  PROC DrawPart72()
    MoveL Offs(pOrigin,295.05,63.65,0.00),v40,z0,tPen\WObj:=wPaper;
    MoveL Offs(pOrigin,298.24,62.80,0.00),v40,z0,tPen\WObj:=wPaper;
    MoveL Offs(pOrigin,301.21,64.85,0.00),v40,z0,tPen\WObj:=wPaper;
    MoveL Offs(pOrigin,304.83,66.20,0.00),v40,z0,tPen\WObj:=wPaper;
    MoveL Offs(pOrigin,310.14,67.40,0.00),v40,z0,tPen\WObj:=wPaper;
    MoveL Offs(pOrigin,314.17,69.95,0.00),v40,z0,tPen\WObj:=wPaper;
    MoveL Offs(pOrigin,316.73,70.95,0.00),v40,z0,tPen\WObj:=wPaper;
    MoveL Offs(pOrigin,322.46,72.57,0.00),v40,z0,tPen\WObj:=wPaper;
    MoveL Offs(pOrigin,333.30,74.49,0.00),v40,z0,tPen\WObj:=wPaper;
    MoveL Offs(pOrigin,334.15,74.91,0.00),v40,z0,tPen\WObj:=wPaper;
    MoveL Offs(pOrigin,334.15,74.91,0.00),v40,z0,tPen\WObj:=wPaper;
    MoveL Offs(pOrigin,340.17,88.09,0.00),v40,z0,tPen\WObj:=wPaper;
    MoveL Offs(pOrigin,342.01,92.97,0.00),v40,z0,tPen\WObj:=wPaper;
    MoveL Offs(pOrigin,341.09,93.74,0.00),v40,z0,tPen\WObj:=wPaper;
    MoveL Offs(pOrigin,345.30,89.53,0.00),v40,z0,tPen\WObj:=wPaper;
    MoveL Offs(pOrigin,344.92,89.84,0.00),v40,z0,tPen\WObj:=wPaper;
    MoveL Offs(pOrigin,341.77,86.69,0.00),v40,fine,tPen\WObj:=wPaper;
    MoveL Offs(pOrigin,341.77,86.69,6.00),v60,z5,tPen\WObj:=wPaper;
    MoveL Offs(pOrigin,339.67,86.08,6.00),vTravel,z5,tPen\WObj:=wPaper;
    MoveL Offs(pOrigin,339.67,86.08,0.00),v60,z0,tPen\WObj:=wPaper;
    MoveL Offs(pOrigin,338.32,84.73,0.00),v40,z0,tPen\WObj:=wPaper;
    MoveL Offs(pOrigin,337.67,85.21,0.00),v40,z0,tPen\WObj:=wPaper;
    MoveL Offs(pOrigin,341.73,81.16,0.00),v40,z0,tPen\WObj:=wPaper;
    MoveL Offs(pOrigin,342.32,82.05,0.00),v40,z0,tPen\WObj:=wPaper;
    MoveL Offs(pOrigin,338.12,86.26,0.00),v40,fine,tPen\WObj:=wPaper;
    MoveL Offs(pOrigin,338.12,86.26,6.00),v60,z5,tPen\WObj:=wPaper;
    MoveL Offs(pOrigin,337.22,84.17,6.00),vTravel,z5,tPen\WObj:=wPaper;
    MoveL Offs(pOrigin,337.22,84.17,0.00),v60,z0,tPen\WObj:=wPaper;
    MoveL Offs(pOrigin,341.28,80.11,0.00),v40,fine,tPen\WObj:=wPaper;
    MoveL Offs(pOrigin,341.28,80.11,6.00),v60,z5,tPen\WObj:=wPaper;
    MoveL Offs(pOrigin,338.14,78.77,6.00),vTravel,z5,tPen\WObj:=wPaper;
    MoveL Offs(pOrigin,338.14,78.77,0.00),v60,z0,tPen\WObj:=wPaper;
    MoveL Offs(pOrigin,345.50,71.41,0.00),v40,fine,tPen\WObj:=wPaper;
    MoveL Offs(pOrigin,345.50,71.41,6.00),v60,z5,tPen\WObj:=wPaper;
    MoveL Offs(pOrigin,343.85,71.56,6.00),vTravel,z5,tPen\WObj:=wPaper;
    MoveL Offs(pOrigin,343.85,71.56,0.00),v60,z0,tPen\WObj:=wPaper;
    MoveL Offs(pOrigin,337.69,77.72,0.00),v40,z0,tPen\WObj:=wPaper;
    MoveL Offs(pOrigin,337.10,76.83,0.00),v40,z0,tPen\WObj:=wPaper;
    MoveL Offs(pOrigin,341.91,72.02,0.00),v40,fine,tPen\WObj:=wPaper;
    MoveL Offs(pOrigin,341.91,72.02,6.00),v60,z5,tPen\WObj:=wPaper;
    MoveL Offs(pOrigin,339.03,73.50,6.00),vTravel,z5,tPen\WObj:=wPaper;
    MoveL Offs(pOrigin,339.03,73.50,0.00),v60,z0,tPen\WObj:=wPaper;
    MoveL Offs(pOrigin,341.89,76.35,0.00),v40,z0,tPen\WObj:=wPaper;
    MoveL Offs(pOrigin,341.89,76.51,0.00),v40,z0,tPen\WObj:=wPaper;
    MoveL Offs(pOrigin,347.45,70.95,0.00),v40,fine,tPen\WObj:=wPaper;
    MoveL Offs(pOrigin,347.45,70.95,6.00),v60,z5,tPen\WObj:=wPaper;
    MoveL Offs(pOrigin,347.44,73.95,6.00),vTravel,z5,tPen\WObj:=wPaper;
    MoveL Offs(pOrigin,347.44,73.95,0.00),v60,z0,tPen\WObj:=wPaper;
    MoveL Offs(pOrigin,344.44,76.95,0.00),v40,fine,tPen\WObj:=wPaper;
    MoveL Offs(pOrigin,344.44,76.95,6.00),v60,z5,tPen\WObj:=wPaper;
    MoveL Offs(pOrigin,345.84,76.25,6.00),vTravel,z5,tPen\WObj:=wPaper;
    MoveL Offs(pOrigin,345.84,76.25,0.00),v60,z0,tPen\WObj:=wPaper;
    MoveL Offs(pOrigin,363.26,76.25,0.00),v40,z0,tPen\WObj:=wPaper;
    MoveL Offs(pOrigin,362.56,76.12,0.00),v40,z0,tPen\WObj:=wPaper;
    MoveL Offs(pOrigin,371.12,84.68,0.00),v40,z0,tPen\WObj:=wPaper;
    MoveL Offs(pOrigin,371.08,84.66,0.00),v40,z0,tPen\WObj:=wPaper;
    MoveL Offs(pOrigin,376.64,79.10,0.00),v40,z0,tPen\WObj:=wPaper;
    MoveL Offs(pOrigin,376.65,79.75,0.00),v40,z0,tPen\WObj:=wPaper;
    MoveL Offs(pOrigin,377.55,80.66,0.00),v40,z0,tPen\WObj:=wPaper;
    MoveL Offs(pOrigin,377.23,81.50,0.00),v40,z0,tPen\WObj:=wPaper;
    MoveL Offs(pOrigin,380.08,78.64,0.00),v40,fine,tPen\WObj:=wPaper;
    MoveL Offs(pOrigin,380.08,78.64,6.00),v60,z5,tPen\WObj:=wPaper;
    MoveL Offs(pOrigin,381.73,78.49,6.00),vTravel,z5,tPen\WObj:=wPaper;
    MoveL Offs(pOrigin,381.73,78.49,0.00),v60,z0,tPen\WObj:=wPaper;
    MoveL Offs(pOrigin,379.18,81.04,0.00),v40,z0,tPen\WObj:=wPaper;
    MoveL Offs(pOrigin,378.90,80.51,0.00),v40,z0,tPen\WObj:=wPaper;
    MoveL Offs(pOrigin,378.00,79.61,0.00),v40,z0,tPen\WObj:=wPaper;
    MoveL Offs(pOrigin,378.29,78.95,0.00),v40,z0,tPen\WObj:=wPaper;
    MoveL Offs(pOrigin,375.73,81.50,0.00),v40,z0,tPen\WObj:=wPaper;
    MoveL Offs(pOrigin,376.35,80.95,0.00),v40,z0,tPen\WObj:=wPaper;
    MoveL Offs(pOrigin,375.15,79.75,0.00),v40,z0,tPen\WObj:=wPaper;
    MoveL Offs(pOrigin,375.14,79.11,0.00),v40,z0,tPen\WObj:=wPaper;
    MoveL Offs(pOrigin,370.03,84.22,0.00),v40,z0,tPen\WObj:=wPaper;
    MoveL Offs(pOrigin,370.91,83.64,0.00),v40,z0,tPen\WObj:=wPaper;
    MoveL Offs(pOrigin,376.65,83.64,0.00),v40,z0,tPen\WObj:=wPaper;
    MoveL Offs(pOrigin,377.56,83.65,0.00),v40,z0,tPen\WObj:=wPaper;
    MoveL Offs(pOrigin,383.12,89.21,0.00),v40,z0,tPen\WObj:=wPaper;
    MoveL Offs(pOrigin,382.45,89.72,0.00),v40,z0,tPen\WObj:=wPaper;
    MoveL Offs(pOrigin,392.06,80.10,0.00),v40,z0,tPen\WObj:=wPaper;
    MoveL Offs(pOrigin,392.53,80.70,0.00),v40,z0,tPen\WObj:=wPaper;
    MoveL Offs(pOrigin,394.03,82.20,0.00),v40,z0,tPen\WObj:=wPaper;
    MoveL Offs(pOrigin,393.44,81.53,0.00),v40,z0,tPen\WObj:=wPaper;
    MoveL Offs(pOrigin,391.10,81.53,0.00),v40,z0,tPen\WObj:=wPaper;
    MoveL Offs(pOrigin,391.48,81.15,0.00),v40,z0,tPen\WObj:=wPaper;
    MoveL Offs(pOrigin,392.99,82.65,0.00),v40,z0,tPen\WObj:=wPaper;
    MoveL Offs(pOrigin,391.94,83.10,0.00),v40,z0,tPen\WObj:=wPaper;
    MoveL Offs(pOrigin,390.44,81.59,0.00),v40,z0,tPen\WObj:=wPaper;
    MoveL Offs(pOrigin,389.66,81.01,0.00),v40,z0,tPen\WObj:=wPaper;
    MoveL Offs(pOrigin,381.40,89.27,0.00),v40,z0,tPen\WObj:=wPaper;
    MoveL Offs(pOrigin,380.35,88.83,0.00),v40,z0,tPen\WObj:=wPaper;
    MoveL Offs(pOrigin,387.41,81.77,0.00),v40,z0,tPen\WObj:=wPaper;
    MoveL Offs(pOrigin,388.04,82.19,0.00),v40,z0,tPen\WObj:=wPaper;
    MoveL Offs(pOrigin,392.40,86.54,0.00),v40,z0,tPen\WObj:=wPaper;
    MoveL Offs(pOrigin,392.94,86.69,0.00),v40,z0,tPen\WObj:=wPaper;
    MoveL Offs(pOrigin,398.05,81.58,0.00),v40,z0,tPen\WObj:=wPaper;
    MoveL Offs(pOrigin,398.53,82.22,0.00),v40,z0,tPen\WObj:=wPaper;
    MoveL Offs(pOrigin,400.03,83.72,0.00),v40,z0,tPen\WObj:=wPaper;
    MoveL Offs(pOrigin,400.14,83.97,0.00),v40,z0,tPen\WObj:=wPaper;
    MoveL Offs(pOrigin,411.86,72.25,0.00),v40,z0,tPen\WObj:=wPaper;
    MoveL Offs(pOrigin,411.50,72.57,0.00),v40,z0,tPen\WObj:=wPaper;
    MoveL Offs(pOrigin,407.67,76.82,0.00),v40,z0,tPen\WObj:=wPaper;
    MoveL Offs(pOrigin,407.60,76.90,0.00),v40,z0,tPen\WObj:=wPaper;
    MoveL Offs(pOrigin,407.60,77.68,0.00),v40,z0,tPen\WObj:=wPaper;
    MoveL Offs(pOrigin,406.61,78.03,0.00),v40,z0,tPen\WObj:=wPaper;
    MoveL Offs(pOrigin,406.40,77.68,0.00),v40,z0,tPen\WObj:=wPaper;
    MoveL Offs(pOrigin,406.61,77.25,0.00),v40,z0,tPen\WObj:=wPaper;
    MoveL Offs(pOrigin,407.60,76.90,0.00),v40,z0,tPen\WObj:=wPaper;
    MoveL Offs(pOrigin,407.35,76.10,0.00),v40,z0,tPen\WObj:=wPaper;
    MoveL Offs(pOrigin,408.40,77.16,0.00),v40,z0,tPen\WObj:=wPaper;
    MoveL Offs(pOrigin,407.80,78.05,0.00),v40,z0,tPen\WObj:=wPaper;
    MoveL Offs(pOrigin,406.45,76.70,0.00),v40,z0,tPen\WObj:=wPaper;
    MoveL Offs(pOrigin,405.85,77.60,0.00),v40,z0,tPen\WObj:=wPaper;
    MoveL Offs(pOrigin,406.91,78.65,0.00),v40,z0,tPen\WObj:=wPaper;
    MoveL Offs(pOrigin,406.16,79.40,0.00),v40,z0,tPen\WObj:=wPaper;
    MoveL Offs(pOrigin,404.96,78.19,0.00),v40,z0,tPen\WObj:=wPaper;
    MoveL Offs(pOrigin,405.12,78.31,0.00),v40,z0,tPen\WObj:=wPaper;
    MoveL Offs(pOrigin,404.70,78.74,0.00),v40,z0,tPen\WObj:=wPaper;
    MoveL Offs(pOrigin,405.12,78.31,0.00),v40,z0,tPen\WObj:=wPaper;
    MoveL Offs(pOrigin,405.76,79.16,0.00),v40,z0,tPen\WObj:=wPaper;
    MoveL Offs(pOrigin,405.55,79.59,0.00),v40,z0,tPen\WObj:=wPaper;
  ENDPROC

  PROC DrawPart73()
    MoveL Offs(pOrigin,405.76,79.16,0.00),v40,z0,tPen\WObj:=wPaper;
    MoveL Offs(pOrigin,404.91,79.42,0.00),v40,z0,tPen\WObj:=wPaper;
    MoveL Offs(pOrigin,403.85,79.42,0.00),v40,z0,tPen\WObj:=wPaper;
    MoveL Offs(pOrigin,404.06,78.79,0.00),v40,z0,tPen\WObj:=wPaper;
    MoveL Offs(pOrigin,405.41,80.14,0.00),v40,z0,tPen\WObj:=wPaper;
    MoveL Offs(pOrigin,404.52,80.74,0.00),v40,z0,tPen\WObj:=wPaper;
    MoveL Offs(pOrigin,403.16,79.39,0.00),v40,z0,tPen\WObj:=wPaper;
    MoveL Offs(pOrigin,402.27,79.98,0.00),v40,z0,tPen\WObj:=wPaper;
    MoveL Offs(pOrigin,403.77,81.49,0.00),v40,z0,tPen\WObj:=wPaper;
    MoveL Offs(pOrigin,403.74,81.86,0.00),v40,z0,tPen\WObj:=wPaper;
    MoveL Offs(pOrigin,416.66,68.94,0.00),v40,z0,tPen\WObj:=wPaper;
    MoveL Offs(pOrigin,416.46,68.79,0.00),v40,z0,tPen\WObj:=wPaper;
    MoveL Offs(pOrigin,412.86,65.19,0.00),v40,z0,tPen\WObj:=wPaper;
    MoveL Offs(pOrigin,413.20,65.35,0.00),v40,z0,tPen\WObj:=wPaper;
    MoveL Offs(pOrigin,412.99,65.78,0.00),v40,z0,tPen\WObj:=wPaper;
    MoveL Offs(pOrigin,413.20,65.35,0.00),v40,z0,tPen\WObj:=wPaper;
    MoveL Offs(pOrigin,412.99,65.69,0.00),v40,z0,tPen\WObj:=wPaper;
    MoveL Offs(pOrigin,415.96,65.69,0.00),v40,z0,tPen\WObj:=wPaper;
    MoveL Offs(pOrigin,415.75,64.63,0.00),v40,z0,tPen\WObj:=wPaper;
    MoveL Offs(pOrigin,413.62,64.63,0.00),v40,z0,tPen\WObj:=wPaper;
    MoveL Offs(pOrigin,413.97,64.50,0.00),v40,z0,tPen\WObj:=wPaper;
    MoveL Offs(pOrigin,413.97,67.69,0.00),v40,z0,tPen\WObj:=wPaper;
    MoveL Offs(pOrigin,412.91,67.90,0.00),v40,z0,tPen\WObj:=wPaper;
    MoveL Offs(pOrigin,412.91,66.62,0.00),v40,z0,tPen\WObj:=wPaper;
    MoveL Offs(pOrigin,412.26,66.08,0.00),v40,z0,tPen\WObj:=wPaper;
    MoveL Offs(pOrigin,416.32,70.14,0.00),v40,z0,tPen\WObj:=wPaper;
    MoveL Offs(pOrigin,416.51,70.59,0.00),v40,z0,tPen\WObj:=wPaper;
    MoveL Offs(pOrigin,411.10,76.00,0.00),v40,z0,tPen\WObj:=wPaper;
    MoveL Offs(pOrigin,411.69,75.97,0.00),v40,z0,tPen\WObj:=wPaper;
    MoveL Offs(pOrigin,413.79,78.07,0.00),v40,z0,tPen\WObj:=wPaper;
    MoveL Offs(pOrigin,414.39,77.19,0.00),v40,z0,tPen\WObj:=wPaper;
    MoveL Offs(pOrigin,408.53,83.05,0.00),v40,z0,tPen\WObj:=wPaper;
    MoveL Offs(pOrigin,409.02,83.75,0.00),v40,z0,tPen\WObj:=wPaper;
    MoveL Offs(pOrigin,410.97,85.70,0.00),v40,z0,tPen\WObj:=wPaper;
    MoveL Offs(pOrigin,410.44,85.75,0.00),v40,z0,tPen\WObj:=wPaper;
    MoveL Offs(pOrigin,408.95,85.75,0.00),v40,z0,tPen\WObj:=wPaper;
    MoveL Offs(pOrigin,408.43,86.14,0.00),v40,z0,tPen\WObj:=wPaper;
    MoveL Offs(pOrigin,410.38,88.10,0.00),v40,z0,tPen\WObj:=wPaper;
    MoveL Offs(pOrigin,410.01,87.86,0.00),v40,z0,tPen\WObj:=wPaper;
    MoveL Offs(pOrigin,408.52,87.86,0.00),v40,z0,tPen\WObj:=wPaper;
    MoveL Offs(pOrigin,408.74,86.81,0.00),v40,z0,tPen\WObj:=wPaper;
    MoveL Offs(pOrigin,410.22,86.81,0.00),v40,z0,tPen\WObj:=wPaper;
    MoveL Offs(pOrigin,410.68,86.90,0.00),v40,z0,tPen\WObj:=wPaper;
    MoveL Offs(pOrigin,408.57,84.80,0.00),v40,z0,tPen\WObj:=wPaper;
    MoveL Offs(pOrigin,409.16,84.70,0.00),v40,z0,tPen\WObj:=wPaper;
    MoveL Offs(pOrigin,410.86,84.70,0.00),v40,z0,tPen\WObj:=wPaper;
    MoveL Offs(pOrigin,411.27,84.50,0.00),v40,z0,tPen\WObj:=wPaper;
    MoveL Offs(pOrigin,409.16,82.40,0.00),v40,z0,tPen\WObj:=wPaper;
    MoveL Offs(pOrigin,409.80,82.58,0.00),v40,z0,tPen\WObj:=wPaper;
    MoveL Offs(pOrigin,411.50,82.58,0.00),v40,z0,tPen\WObj:=wPaper;
    MoveL Offs(pOrigin,411.56,83.31,0.00),v40,z0,tPen\WObj:=wPaper;
    MoveL Offs(pOrigin,409.61,81.35,0.00),v40,z0,tPen\WObj:=wPaper;
    MoveL Offs(pOrigin,409.14,80.95,0.00),v40,z0,tPen\WObj:=wPaper;
    MoveL Offs(pOrigin,415.45,74.64,0.00),v40,z0,tPen\WObj:=wPaper;
    MoveL Offs(pOrigin,415.13,74.93,0.00),v40,z0,tPen\WObj:=wPaper;
    MoveL Offs(pOrigin,413.18,72.98,0.00),v40,z0,tPen\WObj:=wPaper;
    MoveL Offs(pOrigin,412.58,73.87,0.00),v40,z0,tPen\WObj:=wPaper;
    MoveL Offs(pOrigin,414.54,75.83,0.00),v40,fine,tPen\WObj:=wPaper;
    MoveL Offs(pOrigin,414.54,75.83,6.00),v60,z5,tPen\WObj:=wPaper;
    MoveL Offs(pOrigin,414.90,74.14,6.00),vTravel,z5,tPen\WObj:=wPaper;
    MoveL Offs(pOrigin,414.90,74.14,0.00),v60,z0,tPen\WObj:=wPaper;
    MoveL Offs(pOrigin,413.20,74.14,0.00),v40,fine,tPen\WObj:=wPaper;
    MoveL Offs(pOrigin,413.20,74.14,6.00),v60,z5,tPen\WObj:=wPaper;
    MoveL Offs(pOrigin,412.61,71.50,6.00),vTravel,z5,tPen\WObj:=wPaper;
    MoveL Offs(pOrigin,412.61,71.50,0.00),v60,z0,tPen\WObj:=wPaper;
    MoveL Offs(pOrigin,416.67,67.44,0.00),v40,z0,tPen\WObj:=wPaper;
    MoveL Offs(pOrigin,415.96,67.80,0.00),v40,z0,tPen\WObj:=wPaper;
    MoveL Offs(pOrigin,411.50,67.80,0.00),v40,z0,tPen\WObj:=wPaper;
    MoveL Offs(pOrigin,411.07,67.88,0.00),v40,z0,tPen\WObj:=wPaper;
    MoveL Offs(pOrigin,412.87,69.68,0.00),v40,z0,tPen\WObj:=wPaper;
    MoveL Offs(pOrigin,412.49,69.10,0.00),v40,z0,tPen\WObj:=wPaper;
    MoveL Offs(pOrigin,409.80,71.72,0.00),v40,z0,tPen\WObj:=wPaper;
    MoveL Offs(pOrigin,412.49,69.10,0.00),v40,z0,tPen\WObj:=wPaper;
    MoveL Offs(pOrigin,412.78,68.86,0.00),v40,z0,tPen\WObj:=wPaper;
    MoveL Offs(pOrigin,410.65,68.86,0.00),v40,z0,tPen\WObj:=wPaper;
    MoveL Offs(pOrigin,410.47,68.77,0.00),v40,z0,tPen\WObj:=wPaper;
    MoveL Offs(pOrigin,411.97,70.28,0.00),v40,z0,tPen\WObj:=wPaper;
    MoveL Offs(pOrigin,411.71,69.91,0.00),v40,z0,tPen\WObj:=wPaper;
    MoveL Offs(pOrigin,409.59,69.91,0.00),v40,z0,tPen\WObj:=wPaper;
    MoveL Offs(pOrigin,409.80,69.81,0.00),v40,z0,tPen\WObj:=wPaper;
    MoveL Offs(pOrigin,407.89,71.72,0.00),v40,z0,tPen\WObj:=wPaper;
    MoveL Offs(pOrigin,409.80,69.81,0.00),v40,z0,tPen\WObj:=wPaper;
    MoveL Offs(pOrigin,409.57,69.37,0.00),v40,z0,tPen\WObj:=wPaper;
    MoveL Offs(pOrigin,411.38,71.17,0.00),v40,z0,tPen\WObj:=wPaper;
    MoveL Offs(pOrigin,410.65,70.97,0.00),v40,z0,tPen\WObj:=wPaper;
    MoveL Offs(pOrigin,408.52,70.97,0.00),v40,z0,tPen\WObj:=wPaper;
    MoveL Offs(pOrigin,408.08,70.86,0.00),v40,z0,tPen\WObj:=wPaper;
    MoveL Offs(pOrigin,410.03,72.82,0.00),v40,z0,tPen\WObj:=wPaper;
    MoveL Offs(pOrigin,409.59,72.02,0.00),v40,z0,tPen\WObj:=wPaper;
    MoveL Offs(pOrigin,407.46,72.02,0.00),v40,z0,tPen\WObj:=wPaper;
    MoveL Offs(pOrigin,407.33,71.61,0.00),v40,z0,tPen\WObj:=wPaper;
    MoveL Offs(pOrigin,410.19,74.46,0.00),v40,z0,tPen\WObj:=wPaper;
    MoveL Offs(pOrigin,410.01,74.28,0.00),v40,z0,tPen\WObj:=wPaper;
    MoveL Offs(pOrigin,409.38,74.91,0.00),v40,z0,tPen\WObj:=wPaper;
    MoveL Offs(pOrigin,410.01,74.28,0.00),v40,fine,tPen\WObj:=wPaper;
    MoveL Offs(pOrigin,410.01,74.28,6.00),v60,z5,tPen\WObj:=wPaper;
    MoveL Offs(pOrigin,409.74,75.51,6.00),vTravel,z5,tPen\WObj:=wPaper;
    MoveL Offs(pOrigin,409.74,75.51,0.00),v60,z0,tPen\WObj:=wPaper;
    MoveL Offs(pOrigin,406.44,72.21,0.00),v40,z0,tPen\WObj:=wPaper;
    MoveL Offs(pOrigin,406.19,73.08,0.00),v40,z0,tPen\WObj:=wPaper;
    MoveL Offs(pOrigin,408.10,73.08,0.00),v40,fine,tPen\WObj:=wPaper;
    MoveL Offs(pOrigin,408.10,73.08,6.00),v60,z5,tPen\WObj:=wPaper;
    MoveL Offs(pOrigin,407.34,74.61,6.00),vTravel,z5,tPen\WObj:=wPaper;
    MoveL Offs(pOrigin,407.34,74.61,0.00),v60,z0,tPen\WObj:=wPaper;
    MoveL Offs(pOrigin,405.69,72.95,0.00),v40,z0,tPen\WObj:=wPaper;
    MoveL Offs(pOrigin,404.94,73.70,0.00),v40,z0,tPen\WObj:=wPaper;
    MoveL Offs(pOrigin,406.30,75.05,0.00),v40,z0,tPen\WObj:=wPaper;
    MoveL Offs(pOrigin,406.61,74.14,0.00),v40,z0,tPen\WObj:=wPaper;
    MoveL Offs(pOrigin,404.70,74.14,0.00),v40,z0,tPen\WObj:=wPaper;
    MoveL Offs(pOrigin,404.05,74.30,0.00),v40,z0,tPen\WObj:=wPaper;
    MoveL Offs(pOrigin,405.40,75.65,0.00),v40,z0,tPen\WObj:=wPaper;
    MoveL Offs(pOrigin,405.12,75.19,0.00),v40,z0,tPen\WObj:=wPaper;
    MoveL Offs(pOrigin,403.42,75.19,0.00),v40,z0,tPen\WObj:=wPaper;
    MoveL Offs(pOrigin,403.00,74.74,0.00),v40,z0,tPen\WObj:=wPaper;
    MoveL Offs(pOrigin,404.65,76.40,0.00),v40,z0,tPen\WObj:=wPaper;
    MoveL Offs(pOrigin,403.76,76.99,0.00),v40,z0,tPen\WObj:=wPaper;
    MoveL Offs(pOrigin,402.25,75.49,0.00),v40,z0,tPen\WObj:=wPaper;
    MoveL Offs(pOrigin,402.12,74.53,0.00),v40,z0,tPen\WObj:=wPaper;
    MoveL Offs(pOrigin,389.04,87.60,0.00),v40,z0,tPen\WObj:=wPaper;
    MoveL Offs(pOrigin,388.51,87.13,0.00),v40,z0,tPen\WObj:=wPaper;
  ENDPROC

  PROC DrawPart74()
    MoveL Offs(pOrigin,384.45,83.07,0.00),v40,z0,tPen\WObj:=wPaper;
    MoveL Offs(pOrigin,383.52,82.68,0.00),v40,z0,tPen\WObj:=wPaper;
    MoveL Offs(pOrigin,378.56,87.63,0.00),v40,z0,tPen\WObj:=wPaper;
    MoveL Offs(pOrigin,378.35,87.03,0.00),v40,z0,tPen\WObj:=wPaper;
    MoveL Offs(pOrigin,381.75,88.51,0.00),v40,z0,tPen\WObj:=wPaper;
    MoveL Offs(pOrigin,387.06,89.79,0.00),v40,z0,tPen\WObj:=wPaper;
    MoveL Offs(pOrigin,391.10,90.00,0.00),v40,z0,tPen\WObj:=wPaper;
    MoveL Offs(pOrigin,397.05,89.15,0.00),v40,z0,tPen\WObj:=wPaper;
    MoveL Offs(pOrigin,396.68,88.93,0.00),v40,z0,tPen\WObj:=wPaper;
    MoveL Offs(pOrigin,395.63,89.98,0.00),v40,fine,tPen\WObj:=wPaper;
    MoveL Offs(pOrigin,395.63,89.98,6.00),v60,z5,tPen\WObj:=wPaper;
    MoveL Offs(pOrigin,395.78,88.33,6.00),vTravel,z5,tPen\WObj:=wPaper;
    MoveL Offs(pOrigin,395.78,88.33,0.00),v60,z0,tPen\WObj:=wPaper;
    MoveL Offs(pOrigin,393.53,90.58,0.00),v40,fine,tPen\WObj:=wPaper;
    MoveL Offs(pOrigin,393.53,90.58,6.00),v60,z5,tPen\WObj:=wPaper;
    MoveL Offs(pOrigin,391.88,90.74,6.00),vTravel,z5,tPen\WObj:=wPaper;
    MoveL Offs(pOrigin,391.88,90.74,0.00),v60,z0,tPen\WObj:=wPaper;
    MoveL Offs(pOrigin,393.98,88.64,0.00),v40,fine,tPen\WObj:=wPaper;
    MoveL Offs(pOrigin,393.98,88.64,6.00),v60,z5,tPen\WObj:=wPaper;
    MoveL Offs(pOrigin,392.49,88.64,6.00),vTravel,z5,tPen\WObj:=wPaper;
    MoveL Offs(pOrigin,392.49,88.64,0.00),v60,z0,tPen\WObj:=wPaper;
    MoveL Offs(pOrigin,390.38,90.74,0.00),v40,z0,tPen\WObj:=wPaper;
    MoveL Offs(pOrigin,390.16,90.28,0.00),v40,z0,tPen\WObj:=wPaper;
    MoveL Offs(pOrigin,389.26,89.38,0.00),v40,z0,tPen\WObj:=wPaper;
    MoveL Offs(pOrigin,389.49,88.65,0.00),v40,z0,tPen\WObj:=wPaper;
    MoveL Offs(pOrigin,387.39,90.75,0.00),v40,z0,tPen\WObj:=wPaper;
    MoveL Offs(pOrigin,387.17,90.27,0.00),v40,z0,tPen\WObj:=wPaper;
    MoveL Offs(pOrigin,385.82,88.92,0.00),v40,z0,tPen\WObj:=wPaper;
    MoveL Offs(pOrigin,385.22,89.82,0.00),v40,z0,tPen\WObj:=wPaper;
    MoveL Offs(pOrigin,383.87,88.46,0.00),v40,fine,tPen\WObj:=wPaper;
    MoveL Offs(pOrigin,383.87,88.46,6.00),v60,z5,tPen\WObj:=wPaper;
    MoveL Offs(pOrigin,384.16,87.27,6.00),vTravel,z5,tPen\WObj:=wPaper;
    MoveL Offs(pOrigin,384.16,87.27,0.00),v60,z0,tPen\WObj:=wPaper;
    MoveL Offs(pOrigin,380.56,83.66,0.00),v40,z0,tPen\WObj:=wPaper;
    MoveL Offs(pOrigin,380.07,83.14,0.00),v40,z0,tPen\WObj:=wPaper;
    MoveL Offs(pOrigin,376.76,86.44,0.00),v40,z0,tPen\WObj:=wPaper;
    MoveL Offs(pOrigin,377.12,86.20,0.00),v40,z0,tPen\WObj:=wPaper;
    MoveL Offs(pOrigin,373.66,82.74,0.00),v40,z0,tPen\WObj:=wPaper;
    MoveL Offs(pOrigin,374.68,82.55,0.00),v40,z0,tPen\WObj:=wPaper;
    MoveL Offs(pOrigin,372.12,85.11,0.00),v40,z0,tPen\WObj:=wPaper;
    MoveL Offs(pOrigin,373.22,85.29,0.00),v40,z0,tPen\WObj:=wPaper;
    MoveL Offs(pOrigin,367.66,79.73,0.00),v40,z0,tPen\WObj:=wPaper;
    MoveL Offs(pOrigin,367.73,80.01,0.00),v40,z0,tPen\WObj:=wPaper;
    MoveL Offs(pOrigin,371.76,80.44,0.00),v40,z0,tPen\WObj:=wPaper;
    MoveL Offs(pOrigin,377.08,80.44,0.00),v40,z0,tPen\WObj:=wPaper;
    MoveL Offs(pOrigin,383.66,79.16,0.00),v40,z0,tPen\WObj:=wPaper;
    MoveL Offs(pOrigin,387.70,77.68,0.00),v40,z0,tPen\WObj:=wPaper;
    MoveL Offs(pOrigin,386.68,78.02,0.00),v40,z0,tPen\WObj:=wPaper;
    MoveL Offs(pOrigin,385.17,79.53,0.00),v40,fine,tPen\WObj:=wPaper;
    MoveL Offs(pOrigin,385.17,79.53,6.00),v60,z5,tPen\WObj:=wPaper;
    MoveL Offs(pOrigin,385.48,77.73,6.00),vTravel,z5,tPen\WObj:=wPaper;
    MoveL Offs(pOrigin,385.48,77.73,0.00),v60,z0,tPen\WObj:=wPaper;
    MoveL Offs(pOrigin,382.77,80.43,0.00),v40,fine,tPen\WObj:=wPaper;
    MoveL Offs(pOrigin,382.77,80.43,6.00),v60,z5,tPen\WObj:=wPaper;
    MoveL Offs(pOrigin,380.83,80.89,6.00),vTravel,z5,tPen\WObj:=wPaper;
    MoveL Offs(pOrigin,380.83,80.89,0.00),v60,z0,tPen\WObj:=wPaper;
    MoveL Offs(pOrigin,383.68,78.03,0.00),v40,fine,tPen\WObj:=wPaper;
    MoveL Offs(pOrigin,383.68,78.03,6.00),v60,z5,tPen\WObj:=wPaper;
    MoveL Offs(pOrigin,385.47,82.22,6.00),vTravel,z5,tPen\WObj:=wPaper;
    MoveL Offs(pOrigin,385.47,82.22,0.00),v60,z0,tPen\WObj:=wPaper;
    MoveL Offs(pOrigin,379.46,88.23,0.00),v40,z0,tPen\WObj:=wPaper;
    MoveL Offs(pOrigin,379.52,87.10,0.00),v40,z0,tPen\WObj:=wPaper;
    MoveL Offs(pOrigin,375.61,83.20,0.00),v40,z0,tPen\WObj:=wPaper;
    MoveL Offs(pOrigin,376.03,82.70,0.00),v40,z0,tPen\WObj:=wPaper;
    MoveL Offs(pOrigin,373.17,85.55,0.00),v40,fine,tPen\WObj:=wPaper;
    MoveL Offs(pOrigin,373.17,85.55,6.00),v60,z5,tPen\WObj:=wPaper;
    MoveL Offs(pOrigin,374.10,84.70,6.00),vTravel,z5,tPen\WObj:=wPaper;
    MoveL Offs(pOrigin,374.10,84.70,0.00),v60,z0,tPen\WObj:=wPaper;
    MoveL Offs(pOrigin,386.85,84.70,0.00),v40,fine,tPen\WObj:=wPaper;
    MoveL Offs(pOrigin,386.85,84.70,6.00),v60,z5,tPen\WObj:=wPaper;
    MoveL Offs(pOrigin,388.12,83.64,6.00),vTravel,z5,tPen\WObj:=wPaper;
    MoveL Offs(pOrigin,388.12,83.64,0.00),v60,z0,tPen\WObj:=wPaper;
    MoveL Offs(pOrigin,381.75,83.64,0.00),v40,z0,tPen\WObj:=wPaper;
    MoveL Offs(pOrigin,381.75,83.37,0.00),v40,z0,tPen\WObj:=wPaper;
    MoveL Offs(pOrigin,385.66,87.27,0.00),v40,fine,tPen\WObj:=wPaper;
    MoveL Offs(pOrigin,385.66,87.27,6.00),v60,z5,tPen\WObj:=wPaper;
    MoveL Offs(pOrigin,387.16,87.28,6.00),vTravel,z5,tPen\WObj:=wPaper;
    MoveL Offs(pOrigin,387.16,87.28,0.00),v60,z0,tPen\WObj:=wPaper;
    MoveL Offs(pOrigin,383.25,83.37,0.00),v40,z0,tPen\WObj:=wPaper;
    MoveL Offs(pOrigin,383.34,84.48,0.00),v40,z0,tPen\WObj:=wPaper;
    MoveL Offs(pOrigin,383.34,85.96,0.00),v40,z0,tPen\WObj:=wPaper;
    MoveL Offs(pOrigin,382.29,85.96,0.00),v40,z0,tPen\WObj:=wPaper;
    MoveL Offs(pOrigin,382.29,84.48,0.00),v40,z0,tPen\WObj:=wPaper;
    MoveL Offs(pOrigin,381.96,85.11,0.00),v40,z0,tPen\WObj:=wPaper;
    MoveL Offs(pOrigin,384.94,85.11,0.00),v40,z0,tPen\WObj:=wPaper;
    MoveL Offs(pOrigin,384.94,85.11,0.00),v40,z0,tPen\WObj:=wPaper;
    MoveL Offs(pOrigin,389.61,85.32,0.00),v40,z0,tPen\WObj:=wPaper;
    MoveL Offs(pOrigin,393.65,84.47,0.00),v40,z0,tPen\WObj:=wPaper;
    MoveL Offs(pOrigin,398.33,82.85,0.00),v40,z0,tPen\WObj:=wPaper;
    MoveL Offs(pOrigin,401.09,81.36,0.00),v40,z0,tPen\WObj:=wPaper;
    MoveL Offs(pOrigin,405.34,78.38,0.00),v40,z0,tPen\WObj:=wPaper;
    MoveL Offs(pOrigin,405.98,78.38,0.00),v40,z0,tPen\WObj:=wPaper;
    MoveL Offs(pOrigin,405.90,79.16,0.00),v40,z0,tPen\WObj:=wPaper;
    MoveL Offs(pOrigin,403.21,81.29,0.00),v40,z0,tPen\WObj:=wPaper;
    MoveL Offs(pOrigin,402.87,82.08,0.00),v40,z0,tPen\WObj:=wPaper;
    MoveL Offs(pOrigin,401.37,80.58,0.00),v40,z0,tPen\WObj:=wPaper;
    MoveL Offs(pOrigin,402.15,80.47,0.00),v40,z0,tPen\WObj:=wPaper;
    MoveL Offs(pOrigin,403.85,80.47,0.00),v40,z0,tPen\WObj:=wPaper;
    MoveL Offs(pOrigin,404.06,80.65,0.00),v40,z0,tPen\WObj:=wPaper;
    MoveL Offs(pOrigin,404.49,80.44,0.00),v40,z0,tPen\WObj:=wPaper;
    MoveL Offs(pOrigin,404.06,80.65,0.00),v40,fine,tPen\WObj:=wPaper;
    MoveL Offs(pOrigin,404.06,80.65,6.00),v60,z5,tPen\WObj:=wPaper;
    MoveL Offs(pOrigin,401.95,79.17,6.00),vTravel,z5,tPen\WObj:=wPaper;
    MoveL Offs(pOrigin,401.95,79.17,0.00),v60,z0,tPen\WObj:=wPaper;
    MoveL Offs(pOrigin,394.89,86.24,0.00),v40,z0,tPen\WObj:=wPaper;
    MoveL Offs(pOrigin,394.64,85.80,0.00),v40,z0,tPen\WObj:=wPaper;
    MoveL Offs(pOrigin,392.99,84.15,0.00),v40,z0,tPen\WObj:=wPaper;
    MoveL Offs(pOrigin,391.95,84.70,0.00),v40,z0,tPen\WObj:=wPaper;
    MoveL Offs(pOrigin,396.20,84.70,0.00),v40,z0,tPen\WObj:=wPaper;
    MoveL Offs(pOrigin,395.99,85.66,0.00),v40,z0,tPen\WObj:=wPaper;
    MoveL Offs(pOrigin,394.19,83.85,0.00),v40,fine,tPen\WObj:=wPaper;
    MoveL Offs(pOrigin,394.19,83.85,6.00),v60,z5,tPen\WObj:=wPaper;
    MoveL Offs(pOrigin,395.50,82.64,6.00),vTravel,z5,tPen\WObj:=wPaper;
    MoveL Offs(pOrigin,395.50,82.64,0.00),v60,z0,tPen\WObj:=wPaper;
    MoveL Offs(pOrigin,390.99,87.15,0.00),v40,z0,tPen\WObj:=wPaper;
    MoveL Offs(pOrigin,391.20,86.84,0.00),v40,z0,tPen\WObj:=wPaper;
    MoveL Offs(pOrigin,386.99,82.63,0.00),v40,z0,tPen\WObj:=wPaper;
    MoveL Offs(pOrigin,387.91,82.58,0.00),v40,z0,tPen\WObj:=wPaper;
    MoveL Offs(pOrigin,390.89,82.58,0.00),v40,z0,tPen\WObj:=wPaper;
    MoveL Offs(pOrigin,390.89,83.54,0.00),v40,z0,tPen\WObj:=wPaper;
  ENDPROC

  PROC DrawPart75()
    MoveL Offs(pOrigin,389.24,81.89,0.00),v40,fine,tPen\WObj:=wPaper;
    MoveL Offs(pOrigin,389.24,81.89,6.00),v60,z5,tPen\WObj:=wPaper;
    MoveL Offs(pOrigin,391.79,84.44,6.00),vTravel,z5,tPen\WObj:=wPaper;
    MoveL Offs(pOrigin,391.79,84.44,0.00),v60,z0,tPen\WObj:=wPaper;
    MoveL Offs(pOrigin,393.60,86.25,0.00),v40,z0,tPen\WObj:=wPaper;
    MoveL Offs(pOrigin,392.80,85.75,0.00),v40,z0,tPen\WObj:=wPaper;
    MoveL Offs(pOrigin,378.14,85.75,0.00),v40,z0,tPen\WObj:=wPaper;
    MoveL Offs(pOrigin,379.12,85.54,0.00),v40,z0,tPen\WObj:=wPaper;
    MoveL Offs(pOrigin,379.12,84.48,0.00),v40,z0,tPen\WObj:=wPaper;
    MoveL Offs(pOrigin,379.06,83.66,0.00),v40,z0,tPen\WObj:=wPaper;
    MoveL Offs(pOrigin,382.66,87.26,0.00),v40,fine,tPen\WObj:=wPaper;
    MoveL Offs(pOrigin,382.66,87.26,6.00),v60,z5,tPen\WObj:=wPaper;
    MoveL Offs(pOrigin,381.23,85.96,6.00),vTravel,z5,tPen\WObj:=wPaper;
    MoveL Offs(pOrigin,381.23,85.96,0.00),v60,z0,tPen\WObj:=wPaper;
    MoveL Offs(pOrigin,381.23,84.48,0.00),v40,z0,tPen\WObj:=wPaper;
    MoveL Offs(pOrigin,380.17,84.48,0.00),v40,z0,tPen\WObj:=wPaper;
    MoveL Offs(pOrigin,380.17,85.75,0.00),v40,fine,tPen\WObj:=wPaper;
    MoveL Offs(pOrigin,380.17,85.75,6.00),v60,z5,tPen\WObj:=wPaper;
    MoveL Offs(pOrigin,377.66,87.04,6.00),vTravel,z5,tPen\WObj:=wPaper;
    MoveL Offs(pOrigin,377.66,87.04,0.00),v60,z0,tPen\WObj:=wPaper;
    MoveL Offs(pOrigin,381.87,82.83,0.00),v40,fine,tPen\WObj:=wPaper;
    MoveL Offs(pOrigin,381.87,82.83,6.00),v60,z5,tPen\WObj:=wPaper;
    MoveL Offs(pOrigin,378.57,83.14,6.00),vTravel,z5,tPen\WObj:=wPaper;
    MoveL Offs(pOrigin,378.57,83.14,0.00),v60,z0,tPen\WObj:=wPaper;
    MoveL Offs(pOrigin,375.57,86.15,0.00),v40,z0,tPen\WObj:=wPaper;
    MoveL Offs(pOrigin,375.17,85.74,0.00),v40,z0,tPen\WObj:=wPaper;
    MoveL Offs(pOrigin,369.61,80.18,0.00),v40,z0,tPen\WObj:=wPaper;
    MoveL Offs(pOrigin,369.15,79.12,0.00),v40,z0,tPen\WObj:=wPaper;
    MoveL Offs(pOrigin,365.84,82.43,0.00),v40,z0,tPen\WObj:=wPaper;
    MoveL Offs(pOrigin,365.12,81.67,0.00),v40,z0,tPen\WObj:=wPaper;
    MoveL Offs(pOrigin,359.26,75.81,0.00),v40,z0,tPen\WObj:=wPaper;
    MoveL Offs(pOrigin,359.57,75.26,0.00),v40,z0,tPen\WObj:=wPaper;
    MoveL Offs(pOrigin,347.40,87.43,0.00),v40,z0,tPen\WObj:=wPaper;
    MoveL Offs(pOrigin,347.91,88.35,0.00),v40,z0,tPen\WObj:=wPaper;
    MoveL Offs(pOrigin,354.38,94.82,0.00),v40,z0,tPen\WObj:=wPaper;
    MoveL Offs(pOrigin,355.02,94.75,0.00),v40,z0,tPen\WObj:=wPaper;
    MoveL Offs(pOrigin,353.21,96.55,0.00),v40,z0,tPen\WObj:=wPaper;
    MoveL Offs(pOrigin,353.81,97.45,0.00),v40,z0,tPen\WObj:=wPaper;
    MoveL Offs(pOrigin,355.46,95.79,0.00),v40,fine,tPen\WObj:=wPaper;
    MoveL Offs(pOrigin,355.46,95.79,6.00),v60,z5,tPen\WObj:=wPaper;
    MoveL Offs(pOrigin,352.32,94.46,6.00),vTravel,z5,tPen\WObj:=wPaper;
    MoveL Offs(pOrigin,352.32,94.46,0.00),v60,z0,tPen\WObj:=wPaper;
    MoveL Offs(pOrigin,354.43,92.35,0.00),v40,fine,tPen\WObj:=wPaper;
    MoveL Offs(pOrigin,354.43,92.35,6.00),v60,z5,tPen\WObj:=wPaper;
    MoveL Offs(pOrigin,353.98,89.81,6.00),vTravel,z5,tPen\WObj:=wPaper;
    MoveL Offs(pOrigin,353.98,89.81,0.00),v60,z0,tPen\WObj:=wPaper;
    MoveL Offs(pOrigin,343.47,100.33,0.00),v40,fine,tPen\WObj:=wPaper;
    MoveL Offs(pOrigin,343.47,100.33,6.00),v60,z5,tPen\WObj:=wPaper;
    MoveL Offs(pOrigin,343.17,99.13,6.00),vTravel,z5,tPen\WObj:=wPaper;
    MoveL Offs(pOrigin,343.17,99.13,0.00),v60,z0,tPen\WObj:=wPaper;
    MoveL Offs(pOrigin,353.99,88.31,0.00),v40,z0,tPen\WObj:=wPaper;
    MoveL Offs(pOrigin,353.28,88.92,0.00),v40,z0,tPen\WObj:=wPaper;
    MoveL Offs(pOrigin,348.60,88.92,0.00),v40,z0,tPen\WObj:=wPaper;
    MoveL Offs(pOrigin,348.39,87.86,0.00),v40,z0,tPen\WObj:=wPaper;
    MoveL Offs(pOrigin,350.09,87.86,0.00),v40,fine,tPen\WObj:=wPaper;
    MoveL Offs(pOrigin,350.09,87.86,6.00),v60,z5,tPen\WObj:=wPaper;
    MoveL Offs(pOrigin,351.58,86.81,6.00),vTravel,z5,tPen\WObj:=wPaper;
    MoveL Offs(pOrigin,351.58,86.81,0.00),v60,z0,tPen\WObj:=wPaper;
    MoveL Offs(pOrigin,353.28,86.81,0.00),v40,z0,tPen\WObj:=wPaper;
    MoveL Offs(pOrigin,353.60,86.57,0.00),v40,z0,tPen\WObj:=wPaper;
    MoveL Offs(pOrigin,351.20,84.17,0.00),v40,z0,tPen\WObj:=wPaper;
    MoveL Offs(pOrigin,351.79,84.70,0.00),v40,z0,tPen\WObj:=wPaper;
    MoveL Offs(pOrigin,353.28,84.70,0.00),v40,z0,tPen\WObj:=wPaper;
    MoveL Offs(pOrigin,352.72,84.48,0.00),v40,z0,tPen\WObj:=wPaper;
    MoveL Offs(pOrigin,352.72,76.19,0.00),v40,z0,tPen\WObj:=wPaper;
    MoveL Offs(pOrigin,352.97,75.49,0.00),v40,z0,tPen\WObj:=wPaper;
    MoveL Offs(pOrigin,356.12,78.64,0.00),v40,z0,tPen\WObj:=wPaper;
    MoveL Offs(pOrigin,355.40,77.89,0.00),v40,z0,tPen\WObj:=wPaper;
    MoveL Offs(pOrigin,358.80,83.20,0.00),v40,z0,tPen\WObj:=wPaper;
    MoveL Offs(pOrigin,361.99,86.60,0.00),v40,z0,tPen\WObj:=wPaper;
    MoveL Offs(pOrigin,365.81,89.79,0.00),v40,z0,tPen\WObj:=wPaper;
    MoveL Offs(pOrigin,367.94,91.13,0.00),v40,z0,tPen\WObj:=wPaper;
    MoveL Offs(pOrigin,368.79,91.28,0.00),v40,fine,tPen\WObj:=wPaper;
    MoveL Offs(pOrigin,368.79,91.28,6.00),v60,z5,tPen\WObj:=wPaper;
    MoveL Offs(pOrigin,367.32,89.92,6.00),vTravel,z5,tPen\WObj:=wPaper;
    MoveL Offs(pOrigin,367.32,89.92,0.00),v60,z0,tPen\WObj:=wPaper;
    MoveL Offs(pOrigin,366.41,90.82,0.00),v40,z0,tPen\WObj:=wPaper;
    MoveL Offs(pOrigin,365.37,90.37,0.00),v40,z0,tPen\WObj:=wPaper;
    MoveL Offs(pOrigin,366.42,89.32,0.00),v40,z0,tPen\WObj:=wPaper;
    MoveL Offs(pOrigin,365.67,88.57,0.00),v40,z0,tPen\WObj:=wPaper;
    MoveL Offs(pOrigin,364.47,89.77,0.00),v40,z0,tPen\WObj:=wPaper;
    MoveL Offs(pOrigin,363.57,89.18,0.00),v40,z0,tPen\WObj:=wPaper;
    MoveL Offs(pOrigin,364.78,87.98,0.00),v40,z0,tPen\WObj:=wPaper;
    MoveL Offs(pOrigin,364.03,87.23,0.00),v40,z0,tPen\WObj:=wPaper;
    MoveL Offs(pOrigin,360.42,90.84,0.00),v40,z0,tPen\WObj:=wPaper;
    MoveL Offs(pOrigin,360.20,90.19,0.00),v40,z0,tPen\WObj:=wPaper;
    MoveL Offs(pOrigin,363.36,93.35,0.00),v40,z0,tPen\WObj:=wPaper;
    MoveL Offs(pOrigin,363.41,93.82,0.00),v40,z0,tPen\WObj:=wPaper;
    MoveL Offs(pOrigin,365.21,92.02,0.00),v40,z0,tPen\WObj:=wPaper;
    MoveL Offs(pOrigin,365.96,92.77,0.00),v40,z0,tPen\WObj:=wPaper;
    MoveL Offs(pOrigin,364.31,94.42,0.00),v40,z0,tPen\WObj:=wPaper;
    MoveL Offs(pOrigin,365.35,94.87,0.00),v40,z0,tPen\WObj:=wPaper;
    MoveL Offs(pOrigin,366.86,93.36,0.00),v40,z0,tPen\WObj:=wPaper;
    MoveL Offs(pOrigin,367.75,93.96,0.00),v40,z0,tPen\WObj:=wPaper;
    MoveL Offs(pOrigin,366.25,95.46,0.00),v40,z0,tPen\WObj:=wPaper;
    MoveL Offs(pOrigin,366.51,95.00,0.00),v40,z0,tPen\WObj:=wPaper;
    MoveL Offs(pOrigin,360.05,88.54,0.00),v40,z0,tPen\WObj:=wPaper;
    MoveL Offs(pOrigin,360.08,88.94,0.00),v40,z0,tPen\WObj:=wPaper;
    MoveL Offs(pOrigin,361.35,90.21,0.00),v40,z0,tPen\WObj:=wPaper;
    MoveL Offs(pOrigin,360.08,88.94,0.00),v40,fine,tPen\WObj:=wPaper;
    MoveL Offs(pOrigin,360.08,88.94,6.00),v60,z5,tPen\WObj:=wPaper;
    MoveL Offs(pOrigin,358.93,89.34,6.00),vTravel,z5,tPen\WObj:=wPaper;
    MoveL Offs(pOrigin,358.93,89.34,0.00),v60,z0,tPen\WObj:=wPaper;
    MoveL Offs(pOrigin,362.54,85.74,0.00),v40,z0,tPen\WObj:=wPaper;
    MoveL Offs(pOrigin,363.28,86.48,0.00),v40,z0,tPen\WObj:=wPaper;
    MoveL Offs(pOrigin,359.68,90.09,0.00),v40,fine,tPen\WObj:=wPaper;
    MoveL Offs(pOrigin,359.68,90.09,6.00),v60,z5,tPen\WObj:=wPaper;
    MoveL Offs(pOrigin,361.02,91.73,6.00),vTravel,z5,tPen\WObj:=wPaper;
    MoveL Offs(pOrigin,361.02,91.73,0.00),v60,z0,tPen\WObj:=wPaper;
    MoveL Offs(pOrigin,362.67,90.08,0.00),v40,z0,tPen\WObj:=wPaper;
    MoveL Offs(pOrigin,363.42,90.83,0.00),v40,z0,tPen\WObj:=wPaper;
    MoveL Offs(pOrigin,361.92,92.33,0.00),v40,z0,tPen\WObj:=wPaper;
    MoveL Offs(pOrigin,362.51,93.23,0.00),v40,z0,tPen\WObj:=wPaper;
    MoveL Offs(pOrigin,364.32,91.42,0.00),v40,fine,tPen\WObj:=wPaper;
    MoveL Offs(pOrigin,364.32,91.42,6.00),v60,z5,tPen\WObj:=wPaper;
    MoveL Offs(pOrigin,362.29,87.80,6.00),vTravel,z5,tPen\WObj:=wPaper;
    MoveL Offs(pOrigin,362.29,87.80,0.00),v60,z0,tPen\WObj:=wPaper;
    MoveL Offs(pOrigin,358.09,83.59,0.00),v40,z0,tPen\WObj:=wPaper;
    MoveL Offs(pOrigin,357.30,83.51,0.00),v40,z0,tPen\WObj:=wPaper;
    MoveL Offs(pOrigin,359.10,81.70,0.00),v40,z0,tPen\WObj:=wPaper;
  ENDPROC

  PROC DrawPart76()
    MoveL Offs(pOrigin,358.36,80.96,0.00),v40,z0,tPen\WObj:=wPaper;
    MoveL Offs(pOrigin,356.85,82.46,0.00),v40,z0,tPen\WObj:=wPaper;
    MoveL Offs(pOrigin,356.26,81.56,0.00),v40,z0,tPen\WObj:=wPaper;
    MoveL Offs(pOrigin,357.76,80.06,0.00),v40,fine,tPen\WObj:=wPaper;
    MoveL Offs(pOrigin,357.76,80.06,6.00),v60,z5,tPen\WObj:=wPaper;
    MoveL Offs(pOrigin,356.46,80.01,6.00),vTravel,z5,tPen\WObj:=wPaper;
    MoveL Offs(pOrigin,356.46,80.01,0.00),v60,z0,tPen\WObj:=wPaper;
    MoveL Offs(pOrigin,356.67,80.44,0.00),v40,z0,tPen\WObj:=wPaper;
    MoveL Offs(pOrigin,356.46,80.01,0.00),v40,z0,tPen\WObj:=wPaper;
    MoveL Offs(pOrigin,356.28,80.29,0.00),v40,z0,tPen\WObj:=wPaper;
    MoveL Offs(pOrigin,360.64,84.65,0.00),v40,z0,tPen\WObj:=wPaper;
    MoveL Offs(pOrigin,361.19,84.09,0.00),v40,z0,tPen\WObj:=wPaper;
    MoveL Offs(pOrigin,357.89,87.40,0.00),v40,z0,tPen\WObj:=wPaper;
    MoveL Offs(pOrigin,358.48,88.30,0.00),v40,z0,tPen\WObj:=wPaper;
    MoveL Offs(pOrigin,361.79,84.99,0.00),v40,fine,tPen\WObj:=wPaper;
    MoveL Offs(pOrigin,361.79,84.99,6.00),v60,z5,tPen\WObj:=wPaper;
    MoveL Offs(pOrigin,360.45,83.35,6.00),vTravel,z5,tPen\WObj:=wPaper;
    MoveL Offs(pOrigin,360.45,83.35,0.00),v60,z0,tPen\WObj:=wPaper;
    MoveL Offs(pOrigin,357.29,86.50,0.00),v40,fine,tPen\WObj:=wPaper;
    MoveL Offs(pOrigin,357.29,86.50,6.00),v60,z5,tPen\WObj:=wPaper;
    MoveL Offs(pOrigin,356.99,85.30,6.00),vTravel,z5,tPen\WObj:=wPaper;
    MoveL Offs(pOrigin,356.99,85.30,0.00),v60,z0,tPen\WObj:=wPaper;
    MoveL Offs(pOrigin,359.70,82.60,0.00),v40,fine,tPen\WObj:=wPaper;
    MoveL Offs(pOrigin,359.70,82.60,6.00),v60,z5,tPen\WObj:=wPaper;
    MoveL Offs(pOrigin,361.21,79.60,6.00),vTravel,z5,tPen\WObj:=wPaper;
    MoveL Offs(pOrigin,361.21,79.60,0.00),v60,z0,tPen\WObj:=wPaper;
    MoveL Offs(pOrigin,365.41,75.39,0.00),v40,z0,tPen\WObj:=wPaper;
    MoveL Offs(pOrigin,365.55,76.13,0.00),v40,z0,tPen\WObj:=wPaper;
    MoveL Offs(pOrigin,366.91,77.48,0.00),v40,fine,tPen\WObj:=wPaper;
    MoveL Offs(pOrigin,366.91,77.48,6.00),v60,z5,tPen\WObj:=wPaper;
    MoveL Offs(pOrigin,365.71,77.77,6.00),vTravel,z5,tPen\WObj:=wPaper;
    MoveL Offs(pOrigin,365.71,77.77,0.00),v60,z0,tPen\WObj:=wPaper;
    MoveL Offs(pOrigin,364.06,76.12,0.00),v40,z0,tPen\WObj:=wPaper;
    MoveL Offs(pOrigin,363.92,75.40,0.00),v40,z0,tPen\WObj:=wPaper;
    MoveL Offs(pOrigin,360.31,79.00,0.00),v40,z0,tPen\WObj:=wPaper;
    MoveL Offs(pOrigin,360.92,78.36,0.00),v40,z0,tPen\WObj:=wPaper;
    MoveL Offs(pOrigin,364.33,78.36,0.00),v40,z0,tPen\WObj:=wPaper;
    MoveL Offs(pOrigin,364.11,77.30,0.00),v40,z0,tPen\WObj:=wPaper;
    MoveL Offs(pOrigin,351.79,77.30,0.00),v40,z0,tPen\WObj:=wPaper;
    MoveL Offs(pOrigin,350.88,77.98,0.00),v40,z0,tPen\WObj:=wPaper;
    MoveL Offs(pOrigin,354.03,74.83,0.00),v40,z0,tPen\WObj:=wPaper;
    MoveL Offs(pOrigin,354.62,75.64,0.00),v40,z0,tPen\WObj:=wPaper;
    MoveL Offs(pOrigin,357.17,78.20,0.00),v40,fine,tPen\WObj:=wPaper;
    MoveL Offs(pOrigin,357.17,78.20,6.00),v60,z5,tPen\WObj:=wPaper;
    MoveL Offs(pOrigin,358.97,78.50,6.00),vTravel,z5,tPen\WObj:=wPaper;
    MoveL Offs(pOrigin,358.97,78.50,0.00),v60,z0,tPen\WObj:=wPaper;
    MoveL Offs(pOrigin,356.11,75.65,0.00),v40,z0,tPen\WObj:=wPaper;
    MoveL Offs(pOrigin,356.58,75.27,0.00),v40,z0,tPen\WObj:=wPaper;
    MoveL Offs(pOrigin,347.26,84.58,0.00),v40,z0,tPen\WObj:=wPaper;
    MoveL Offs(pOrigin,348.17,84.70,0.00),v40,z0,tPen\WObj:=wPaper;
    MoveL Offs(pOrigin,349.66,84.70,0.00),v40,z0,tPen\WObj:=wPaper;
    MoveL Offs(pOrigin,349.45,83.64,0.00),v40,z0,tPen\WObj:=wPaper;
    MoveL Offs(pOrigin,348.17,83.64,0.00),v40,fine,tPen\WObj:=wPaper;
    MoveL Offs(pOrigin,348.17,83.64,6.00),v60,z5,tPen\WObj:=wPaper;
    MoveL Offs(pOrigin,347.26,86.08,6.00),vTravel,z5,tPen\WObj:=wPaper;
    MoveL Offs(pOrigin,347.26,86.08,0.00),v60,z0,tPen\WObj:=wPaper;
    MoveL Offs(pOrigin,358.07,75.26,0.00),v40,z0,tPen\WObj:=wPaper;
    MoveL Offs(pOrigin,357.76,75.80,0.00),v40,z0,tPen\WObj:=wPaper;
    MoveL Offs(pOrigin,361.52,79.56,0.00),v40,z0,tPen\WObj:=wPaper;
    MoveL Offs(pOrigin,362.25,80.04,0.00),v40,z0,tPen\WObj:=wPaper;
    MoveL Offs(pOrigin,367.06,75.24,0.00),v40,z0,tPen\WObj:=wPaper;
    MoveL Offs(pOrigin,366.90,75.98,0.00),v40,z0,tPen\WObj:=wPaper;
    MoveL Offs(pOrigin,368.25,77.33,0.00),v40,z0,tPen\WObj:=wPaper;
    MoveL Offs(pOrigin,369.15,77.63,0.00),v40,z0,tPen\WObj:=wPaper;
    MoveL Offs(pOrigin,371.86,74.92,0.00),v40,z0,tPen\WObj:=wPaper;
    MoveL Offs(pOrigin,372.44,75.55,0.00),v40,z0,tPen\WObj:=wPaper;
    MoveL Offs(pOrigin,373.19,76.30,0.00),v40,z0,tPen\WObj:=wPaper;
    MoveL Offs(pOrigin,372.75,77.02,0.00),v40,z0,tPen\WObj:=wPaper;
    MoveL Offs(pOrigin,375.75,74.01,0.00),v40,fine,tPen\WObj:=wPaper;
    MoveL Offs(pOrigin,375.75,74.01,6.00),v60,z5,tPen\WObj:=wPaper;
    MoveL Offs(pOrigin,376.95,75.81,6.00),vTravel,z5,tPen\WObj:=wPaper;
    MoveL Offs(pOrigin,376.95,75.81,0.00),v60,z0,tPen\WObj:=wPaper;
    MoveL Offs(pOrigin,380.85,71.90,0.00),v40,fine,tPen\WObj:=wPaper;
    MoveL Offs(pOrigin,380.85,71.90,6.00),v60,z5,tPen\WObj:=wPaper;
    MoveL Offs(pOrigin,382.05,73.69,6.00),vTravel,z5,tPen\WObj:=wPaper;
    MoveL Offs(pOrigin,382.05,73.69,0.00),v60,z0,tPen\WObj:=wPaper;
    MoveL Offs(pOrigin,400.08,55.66,0.00),v40,fine,tPen\WObj:=wPaper;
    MoveL Offs(pOrigin,400.08,55.66,6.00),v60,z5,tPen\WObj:=wPaper;
    MoveL Offs(pOrigin,398.33,56.42,6.00),vTravel,z5,tPen\WObj:=wPaper;
    MoveL Offs(pOrigin,398.33,56.42,0.00),v60,z0,tPen\WObj:=wPaper;
    MoveL Offs(pOrigin,398.11,56.85,0.00),v40,z0,tPen\WObj:=wPaper;
    MoveL Offs(pOrigin,398.33,56.42,0.00),v40,fine,tPen\WObj:=wPaper;
    MoveL Offs(pOrigin,398.33,56.42,6.00),v60,z5,tPen\WObj:=wPaper;
    MoveL Offs(pOrigin,397.69,57.49,6.00),vTravel,z5,tPen\WObj:=wPaper;
    MoveL Offs(pOrigin,397.69,57.49,0.00),v60,z0,tPen\WObj:=wPaper;
    MoveL Offs(pOrigin,397.26,58.12,0.00),v40,z0,tPen\WObj:=wPaper;
    MoveL Offs(pOrigin,397.69,57.49,0.00),v40,fine,tPen\WObj:=wPaper;
    MoveL Offs(pOrigin,397.69,57.49,6.00),v60,z5,tPen\WObj:=wPaper;
    MoveL Offs(pOrigin,396.84,58.76,6.00),vTravel,z5,tPen\WObj:=wPaper;
    MoveL Offs(pOrigin,396.84,58.76,0.00),v60,z0,tPen\WObj:=wPaper;
    MoveL Offs(pOrigin,396.41,59.40,0.00),v40,z0,tPen\WObj:=wPaper;
    MoveL Offs(pOrigin,396.84,58.76,0.00),v40,z0,tPen\WObj:=wPaper;
    MoveL Offs(pOrigin,395.72,58.52,0.00),v40,z0,tPen\WObj:=wPaper;
    MoveL Offs(pOrigin,401.13,53.11,0.00),v40,fine,tPen\WObj:=wPaper;
    MoveL Offs(pOrigin,401.13,53.11,6.00),v60,z5,tPen\WObj:=wPaper;
    MoveL Offs(pOrigin,399.81,53.66,6.00),vTravel,z5,tPen\WObj:=wPaper;
    MoveL Offs(pOrigin,399.81,53.66,0.00),v60,z0,tPen\WObj:=wPaper;
    MoveL Offs(pOrigin,399.60,54.09,0.00),v40,z0,tPen\WObj:=wPaper;
    MoveL Offs(pOrigin,399.81,53.66,0.00),v40,fine,tPen\WObj:=wPaper;
    MoveL Offs(pOrigin,399.81,53.66,6.00),v60,z5,tPen\WObj:=wPaper;
    MoveL Offs(pOrigin,398.28,54.47,6.00),vTravel,z5,tPen\WObj:=wPaper;
    MoveL Offs(pOrigin,398.28,54.47,0.00),v60,z0,tPen\WObj:=wPaper;
    MoveL Offs(pOrigin,401.89,50.86,0.00),v40,fine,tPen\WObj:=wPaper;
    MoveL Offs(pOrigin,401.89,50.86,6.00),v60,z5,tPen\WObj:=wPaper;
    MoveL Offs(pOrigin,400.40,49.37,6.00),vTravel,z5,tPen\WObj:=wPaper;
    MoveL Offs(pOrigin,400.40,49.37,0.00),v60,z0,tPen\WObj:=wPaper;
    MoveL Offs(pOrigin,402.80,46.96,0.00),v40,fine,tPen\WObj:=wPaper;
    MoveL Offs(pOrigin,402.80,46.96,6.00),v60,z5,tPen\WObj:=wPaper;
    MoveL Offs(pOrigin,402.81,45.47,6.00),vTravel,z5,tPen\WObj:=wPaper;
    MoveL Offs(pOrigin,402.81,45.47,0.00),v60,z0,tPen\WObj:=wPaper;
    MoveL Offs(pOrigin,401.00,47.27,0.00),v40,fine,tPen\WObj:=wPaper;
    MoveL Offs(pOrigin,401.00,47.27,6.00),v60,z5,tPen\WObj:=wPaper;
    MoveL Offs(pOrigin,401.46,45.32,6.00),vTravel,z5,tPen\WObj:=wPaper;
    MoveL Offs(pOrigin,401.46,45.32,0.00),v60,z0,tPen\WObj:=wPaper;
    MoveL Offs(pOrigin,402.66,44.12,0.00),v40,fine,tPen\WObj:=wPaper;
    MoveL Offs(pOrigin,402.66,44.12,6.00),v60,z5,tPen\WObj:=wPaper;
    MoveL Offs(pOrigin,402.58,42.19,6.00),vTravel,z5,tPen\WObj:=wPaper;
    MoveL Offs(pOrigin,402.58,42.19,0.00),v60,z0,tPen\WObj:=wPaper;
    MoveL Offs(pOrigin,401.94,47.71,0.00),v40,z0,tPen\WObj:=wPaper;
    MoveL Offs(pOrigin,399.88,53.88,0.00),v40,z0,tPen\WObj:=wPaper;
  ENDPROC

  PROC DrawPart77()
    MoveL Offs(pOrigin,396.20,60.04,0.00),v40,z0,tPen\WObj:=wPaper;
    MoveL Offs(pOrigin,392.59,64.50,0.00),v40,z0,tPen\WObj:=wPaper;
    MoveL Offs(pOrigin,387.91,68.75,0.00),v40,z0,tPen\WObj:=wPaper;
    MoveL Offs(pOrigin,382.81,72.22,0.00),v40,z0,tPen\WObj:=wPaper;
    MoveL Offs(pOrigin,377.08,74.77,0.00),v40,z0,tPen\WObj:=wPaper;
    MoveL Offs(pOrigin,370.49,76.40,0.00),v40,z0,tPen\WObj:=wPaper;
    MoveL Offs(pOrigin,370.42,76.19,0.00),v40,z0,tPen\WObj:=wPaper;
    MoveL Offs(pOrigin,369.64,75.97,0.00),v40,z0,tPen\WObj:=wPaper;
    MoveL Offs(pOrigin,369.00,76.61,0.00),v40,z0,tPen\WObj:=wPaper;
    MoveL Offs(pOrigin,369.85,76.82,0.00),v40,z0,tPen\WObj:=wPaper;
    MoveL Offs(pOrigin,370.42,76.19,0.00),v40,z0,tPen\WObj:=wPaper;
    MoveL Offs(pOrigin,370.80,76.89,0.00),v40,z0,tPen\WObj:=wPaper;
    MoveL Offs(pOrigin,369.60,75.69,0.00),v40,z0,tPen\WObj:=wPaper;
    MoveL Offs(pOrigin,370.21,75.08,0.00),v40,z0,tPen\WObj:=wPaper;
    MoveL Offs(pOrigin,363.90,81.39,0.00),v40,z0,tPen\WObj:=wPaper;
    MoveL Offs(pOrigin,363.15,80.64,0.00),v40,z0,tPen\WObj:=wPaper;
    MoveL Offs(pOrigin,368.56,75.23,0.00),v40,z0,tPen\WObj:=wPaper;
    MoveL Offs(pOrigin,368.40,75.98,0.00),v40,z0,tPen\WObj:=wPaper;
    MoveL Offs(pOrigin,369.45,77.04,0.00),v40,fine,tPen\WObj:=wPaper;
    MoveL Offs(pOrigin,369.45,77.04,6.00),v60,z5,tPen\WObj:=wPaper;
    MoveL Offs(pOrigin,370.95,77.32,6.00),vTravel,z5,tPen\WObj:=wPaper;
    MoveL Offs(pOrigin,370.95,77.32,0.00),v60,z0,tPen\WObj:=wPaper;
    MoveL Offs(pOrigin,373.65,74.62,0.00),v40,fine,tPen\WObj:=wPaper;
    MoveL Offs(pOrigin,373.65,74.62,6.00),v60,z5,tPen\WObj:=wPaper;
    MoveL Offs(pOrigin,374.85,76.41,6.00),vTravel,z5,tPen\WObj:=wPaper;
    MoveL Offs(pOrigin,374.85,76.41,0.00),v60,z0,tPen\WObj:=wPaper;
    MoveL Offs(pOrigin,378.15,73.11,0.00),v40,fine,tPen\WObj:=wPaper;
    MoveL Offs(pOrigin,378.15,73.11,6.00),v60,z5,tPen\WObj:=wPaper;
    MoveL Offs(pOrigin,379.05,75.20,6.00),vTravel,z5,tPen\WObj:=wPaper;
    MoveL Offs(pOrigin,379.05,75.20,0.00),v60,z0,tPen\WObj:=wPaper;
    MoveL Offs(pOrigin,384.76,69.49,0.00),v40,z0,tPen\WObj:=wPaper;
    MoveL Offs(pOrigin,385.91,69.60,0.00),v40,z0,tPen\WObj:=wPaper;
    MoveL Offs(pOrigin,386.66,70.35,0.00),v40,fine,tPen\WObj:=wPaper;
    MoveL Offs(pOrigin,386.66,70.35,6.00),v60,z5,tPen\WObj:=wPaper;
    MoveL Offs(pOrigin,385.50,71.73,6.00),vTravel,z5,tPen\WObj:=wPaper;
    MoveL Offs(pOrigin,385.50,71.73,0.00),v60,z0,tPen\WObj:=wPaper;
    MoveL Offs(pOrigin,397.82,59.41,0.00),v40,fine,tPen\WObj:=wPaper;
    MoveL Offs(pOrigin,397.82,59.41,6.00),v60,z5,tPen\WObj:=wPaper;
    MoveL Offs(pOrigin,395.56,60.67,6.00),vTravel,z5,tPen\WObj:=wPaper;
    MoveL Offs(pOrigin,395.56,60.67,0.00),v60,z0,tPen\WObj:=wPaper;
    MoveL Offs(pOrigin,395.14,61.10,0.00),v40,z0,tPen\WObj:=wPaper;
    MoveL Offs(pOrigin,395.56,60.67,0.00),v40,fine,tPen\WObj:=wPaper;
    MoveL Offs(pOrigin,395.56,60.67,6.00),v60,z5,tPen\WObj:=wPaper;
    MoveL Offs(pOrigin,394.29,62.16,6.00),vTravel,z5,tPen\WObj:=wPaper;
    MoveL Offs(pOrigin,394.29,62.16,0.00),v60,z0,tPen\WObj:=wPaper;
    MoveL Offs(pOrigin,393.86,62.80,0.00),v40,z0,tPen\WObj:=wPaper;
    MoveL Offs(pOrigin,394.29,62.16,0.00),v40,fine,tPen\WObj:=wPaper;
    MoveL Offs(pOrigin,394.29,62.16,6.00),v60,z5,tPen\WObj:=wPaper;
    MoveL Offs(pOrigin,393.44,63.22,6.00),vTravel,z5,tPen\WObj:=wPaper;
    MoveL Offs(pOrigin,393.44,63.22,0.00),v60,z0,tPen\WObj:=wPaper;
    MoveL Offs(pOrigin,393.01,63.65,0.00),v40,z0,tPen\WObj:=wPaper;
    MoveL Offs(pOrigin,393.44,63.22,0.00),v40,fine,tPen\WObj:=wPaper;
    MoveL Offs(pOrigin,393.44,63.22,6.00),v60,z5,tPen\WObj:=wPaper;
    MoveL Offs(pOrigin,392.18,63.92,6.00),vTravel,z5,tPen\WObj:=wPaper;
    MoveL Offs(pOrigin,392.18,63.92,0.00),v60,z0,tPen\WObj:=wPaper;
    MoveL Offs(pOrigin,392.93,64.67,0.00),v40,z0,tPen\WObj:=wPaper;
    MoveL Offs(pOrigin,392.16,64.71,0.00),v40,z0,tPen\WObj:=wPaper;
    MoveL Offs(pOrigin,391.52,65.35,0.00),v40,z0,tPen\WObj:=wPaper;
    MoveL Offs(pOrigin,392.16,64.71,0.00),v40,fine,tPen\WObj:=wPaper;
    MoveL Offs(pOrigin,392.16,64.71,6.00),v60,z5,tPen\WObj:=wPaper;
    MoveL Offs(pOrigin,391.31,65.56,6.00),vTravel,z5,tPen\WObj:=wPaper;
    MoveL Offs(pOrigin,391.31,65.56,0.00),v60,z0,tPen\WObj:=wPaper;
    MoveL Offs(pOrigin,390.67,66.20,0.00),v40,z0,tPen\WObj:=wPaper;
    MoveL Offs(pOrigin,391.31,65.56,0.00),v40,z0,tPen\WObj:=wPaper;
    MoveL Offs(pOrigin,391.44,66.17,0.00),v40,z0,tPen\WObj:=wPaper;
    MoveL Offs(pOrigin,390.69,65.42,0.00),v40,fine,tPen\WObj:=wPaper;
    MoveL Offs(pOrigin,390.69,65.42,6.00),v60,z5,tPen\WObj:=wPaper;
    MoveL Offs(pOrigin,389.61,67.05,6.00),vTravel,z5,tPen\WObj:=wPaper;
    MoveL Offs(pOrigin,389.61,67.05,0.00),v60,z0,tPen\WObj:=wPaper;
    MoveL Offs(pOrigin,388.98,67.69,0.00),v40,z0,tPen\WObj:=wPaper;
    MoveL Offs(pOrigin,389.61,67.05,0.00),v40,fine,tPen\WObj:=wPaper;
    MoveL Offs(pOrigin,389.61,67.05,6.00),v60,z5,tPen\WObj:=wPaper;
    MoveL Offs(pOrigin,388.30,69.00,6.00),vTravel,z5,tPen\WObj:=wPaper;
    MoveL Offs(pOrigin,388.30,69.00,0.00),v60,z0,tPen\WObj:=wPaper;
    MoveL Offs(pOrigin,387.55,68.25,0.00),v40,fine,tPen\WObj:=wPaper;
    MoveL Offs(pOrigin,387.55,68.25,6.00),v60,z5,tPen\WObj:=wPaper;
    MoveL Offs(pOrigin,394.76,78.90,6.00),vTravel,z5,tPen\WObj:=wPaper;
    MoveL Offs(pOrigin,394.76,78.90,0.00),v60,z0,tPen\WObj:=wPaper;
    MoveL Offs(pOrigin,383.64,90.02,0.00),v40,fine,tPen\WObj:=wPaper;
    MoveL Offs(pOrigin,383.64,90.02,6.00),v60,z5,tPen\WObj:=wPaper;
    MoveL Offs(pOrigin,384.84,90.31,6.00),vTravel,z5,tPen\WObj:=wPaper;
    MoveL Offs(pOrigin,384.84,90.31,0.00),v60,z0,tPen\WObj:=wPaper;
    MoveL Offs(pOrigin,397.76,77.39,0.00),v40,z0,tPen\WObj:=wPaper;
    MoveL Offs(pOrigin,398.51,77.72,0.00),v40,z0,tPen\WObj:=wPaper;
    MoveL Offs(pOrigin,400.02,79.23,0.00),v40,z0,tPen\WObj:=wPaper;
    MoveL Offs(pOrigin,400.15,79.48,0.00),v40,z0,tPen\WObj:=wPaper;
    MoveL Offs(pOrigin,416.53,63.10,0.00),v40,z0,tPen\WObj:=wPaper;
    MoveL Offs(pOrigin,416.44,62.80,0.00),v40,z0,tPen\WObj:=wPaper;
    MoveL Offs(pOrigin,414.19,60.55,0.00),v40,z0,tPen\WObj:=wPaper;
    MoveL Offs(pOrigin,414.69,60.41,0.00),v40,z0,tPen\WObj:=wPaper;
    MoveL Offs(pOrigin,416.17,60.41,0.00),v40,z0,tPen\WObj:=wPaper;
    MoveL Offs(pOrigin,416.74,60.10,0.00),v40,z0,tPen\WObj:=wPaper;
    MoveL Offs(pOrigin,414.33,57.70,0.00),v40,z0,tPen\WObj:=wPaper;
    MoveL Offs(pOrigin,414.00,58.17,0.00),v40,z0,tPen\WObj:=wPaper;
    MoveL Offs(pOrigin,417.46,54.71,0.00),v40,fine,tPen\WObj:=wPaper;
    MoveL Offs(pOrigin,417.46,54.71,6.00),v60,z5,tPen\WObj:=wPaper;
    MoveL Offs(pOrigin,417.45,56.21,6.00),vTravel,z5,tPen\WObj:=wPaper;
    MoveL Offs(pOrigin,417.45,56.21,0.00),v60,z0,tPen\WObj:=wPaper;
    MoveL Offs(pOrigin,413.70,59.96,0.00),v40,z0,tPen\WObj:=wPaper;
    MoveL Offs(pOrigin,414.19,59.05,0.00),v40,z0,tPen\WObj:=wPaper;
    MoveL Offs(pOrigin,416.59,61.45,0.00),v40,z0,tPen\WObj:=wPaper;
    MoveL Offs(pOrigin,415.96,61.46,0.00),v40,z0,tPen\WObj:=wPaper;
    MoveL Offs(pOrigin,414.48,61.46,0.00),v40,z0,tPen\WObj:=wPaper;
    MoveL Offs(pOrigin,415.02,60.89,0.00),v40,z0,tPen\WObj:=wPaper;
    MoveL Offs(pOrigin,415.02,71.51,0.00),v40,fine,tPen\WObj:=wPaper;
    MoveL Offs(pOrigin,415.02,71.51,6.00),v60,z5,tPen\WObj:=wPaper;
    MoveL Offs(pOrigin,416.05,72.54,6.00),vTravel,z5,tPen\WObj:=wPaper;
    MoveL Offs(pOrigin,416.05,72.54,0.00),v60,z0,tPen\WObj:=wPaper;
    MoveL Offs(pOrigin,410.04,78.55,0.00),v40,z0,tPen\WObj:=wPaper;
    MoveL Offs(pOrigin,410.50,79.26,0.00),v40,z0,tPen\WObj:=wPaper;
    MoveL Offs(pOrigin,412.46,81.21,0.00),v40,z0,tPen\WObj:=wPaper;
    MoveL Offs(pOrigin,411.71,81.53,0.00),v40,z0,tPen\WObj:=wPaper;
    MoveL Offs(pOrigin,410.22,81.53,0.00),v40,z0,tPen\WObj:=wPaper;
    MoveL Offs(pOrigin,410.80,81.29,0.00),v40,z0,tPen\WObj:=wPaper;
    MoveL Offs(pOrigin,410.80,82.99,0.00),v40,z0,tPen\WObj:=wPaper;
    MoveL Offs(pOrigin,411.08,83.64,0.00),v40,z0,tPen\WObj:=wPaper;
    MoveL Offs(pOrigin,409.59,83.64,0.00),v40,z0,tPen\WObj:=wPaper;
    MoveL Offs(pOrigin,409.74,84.69,0.00),v40,z0,tPen\WObj:=wPaper;
    MoveL Offs(pOrigin,409.74,86.60,0.00),v40,fine,tPen\WObj:=wPaper;
    MoveL Offs(pOrigin,409.74,86.60,6.00),v60,z5,tPen\WObj:=wPaper;
  ENDPROC

  PROC DrawPart78()
    MoveL Offs(pOrigin,411.52,86.04,6.00),vTravel,z5,tPen\WObj:=wPaper;
    MoveL Offs(pOrigin,411.52,86.04,0.00),v60,z0,tPen\WObj:=wPaper;
    MoveL Offs(pOrigin,406.71,90.84,0.00),v40,z0,tPen\WObj:=wPaper;
    MoveL Offs(pOrigin,407.09,90.78,0.00),v40,z0,tPen\WObj:=wPaper;
    MoveL Offs(pOrigin,409.20,92.89,0.00),v40,z0,tPen\WObj:=wPaper;
    MoveL Offs(pOrigin,408.74,93.14,0.00),v40,z0,tPen\WObj:=wPaper;
    MoveL Offs(pOrigin,407.25,93.14,0.00),v40,z0,tPen\WObj:=wPaper;
    MoveL Offs(pOrigin,407.63,93.61,0.00),v40,z0,tPen\WObj:=wPaper;
    MoveL Offs(pOrigin,407.63,94.89,0.00),v40,z0,tPen\WObj:=wPaper;
    MoveL Offs(pOrigin,408.10,95.26,0.00),v40,z0,tPen\WObj:=wPaper;
    MoveL Offs(pOrigin,406.61,95.26,0.00),v40,z0,tPen\WObj:=wPaper;
    MoveL Offs(pOrigin,405.91,95.57,0.00),v40,z0,tPen\WObj:=wPaper;
    MoveL Offs(pOrigin,407.86,97.53,0.00),v40,z0,tPen\WObj:=wPaper;
    MoveL Offs(pOrigin,407.25,97.37,0.00),v40,z0,tPen\WObj:=wPaper;
    MoveL Offs(pOrigin,405.76,97.37,0.00),v40,z0,tPen\WObj:=wPaper;
    MoveL Offs(pOrigin,405.46,96.62,0.00),v40,z0,tPen\WObj:=wPaper;
    MoveL Offs(pOrigin,407.42,98.57,0.00),v40,z0,tPen\WObj:=wPaper;
    MoveL Offs(pOrigin,407.89,98.63,0.00),v40,z0,tPen\WObj:=wPaper;
    MoveL Offs(pOrigin,395.86,110.65,0.00),v40,z0,tPen\WObj:=wPaper;
    MoveL Offs(pOrigin,395.32,110.37,0.00),v40,z0,tPen\WObj:=wPaper;
    MoveL Offs(pOrigin,393.97,109.02,0.00),v40,z0,tPen\WObj:=wPaper;
    MoveL Offs(pOrigin,393.32,108.71,0.00),v40,z0,tPen\WObj:=wPaper;
    MoveL Offs(pOrigin,388.82,113.22,0.00),v40,fine,tPen\WObj:=wPaper;
    MoveL Offs(pOrigin,388.82,113.22,6.00),v60,z5,tPen\WObj:=wPaper;
    MoveL Offs(pOrigin,389.78,112.30,6.00),vTravel,z5,tPen\WObj:=wPaper;
    MoveL Offs(pOrigin,389.78,112.30,0.00),v60,z0,tPen\WObj:=wPaper;
    MoveL Offs(pOrigin,389.03,111.55,0.00),v40,z0,tPen\WObj:=wPaper;
    MoveL Offs(pOrigin,388.07,110.97,0.00),v40,z0,tPen\WObj:=wPaper;
    MoveL Offs(pOrigin,385.22,113.83,0.00),v40,fine,tPen\WObj:=wPaper;
    MoveL Offs(pOrigin,385.22,113.83,6.00),v60,z5,tPen\WObj:=wPaper;
    MoveL Offs(pOrigin,383.72,113.83,6.00),vTravel,z5,tPen\WObj:=wPaper;
    MoveL Offs(pOrigin,383.72,113.83,0.00),v60,z0,tPen\WObj:=wPaper;
    MoveL Offs(pOrigin,385.67,111.88,0.00),v40,fine,tPen\WObj:=wPaper;
    MoveL Offs(pOrigin,385.67,111.88,6.00),v60,z5,tPen\WObj:=wPaper;
    MoveL Offs(pOrigin,387.02,113.52,6.00),vTravel,z5,tPen\WObj:=wPaper;
    MoveL Offs(pOrigin,387.02,113.52,0.00),v60,z0,tPen\WObj:=wPaper;
    MoveL Offs(pOrigin,390.47,110.07,0.00),v40,z0,tPen\WObj:=wPaper;
    MoveL Offs(pOrigin,391.13,110.66,0.00),v40,z0,tPen\WObj:=wPaper;
    MoveL Offs(pOrigin,392.03,111.56,0.00),v40,z0,tPen\WObj:=wPaper;
    MoveL Offs(pOrigin,391.10,111.46,0.00),v40,z0,tPen\WObj:=wPaper;
    MoveL Offs(pOrigin,386.42,112.74,0.00),v40,z0,tPen\WObj:=wPaper;
    MoveL Offs(pOrigin,381.96,113.38,0.00),v40,z0,tPen\WObj:=wPaper;
    MoveL Offs(pOrigin,382.82,113.24,0.00),v40,z0,tPen\WObj:=wPaper;
    MoveL Offs(pOrigin,383.58,112.49,0.00),v40,fine,tPen\WObj:=wPaper;
    MoveL Offs(pOrigin,383.58,112.49,6.00),v60,z5,tPen\WObj:=wPaper;
    MoveL Offs(pOrigin,382.54,109.04,6.00),vTravel,z5,tPen\WObj:=wPaper;
    MoveL Offs(pOrigin,382.54,109.04,0.00),v60,z0,tPen\WObj:=wPaper;
    MoveL Offs(pOrigin,385.39,106.19,0.00),v40,fine,tPen\WObj:=wPaper;
    MoveL Offs(pOrigin,385.39,106.19,6.00),v60,z5,tPen\WObj:=wPaper;
    MoveL Offs(pOrigin,385.10,104.99,6.00),vTravel,z5,tPen\WObj:=wPaper;
    MoveL Offs(pOrigin,385.10,104.99,0.00),v60,z0,tPen\WObj:=wPaper;
    MoveL Offs(pOrigin,389.00,101.08,0.00),v40,z0,tPen\WObj:=wPaper;
    MoveL Offs(pOrigin,389.60,101.66,0.00),v40,z0,tPen\WObj:=wPaper;
    MoveL Offs(pOrigin,390.80,102.87,0.00),v40,z0,tPen\WObj:=wPaper;
    MoveL Offs(pOrigin,391.09,103.47,0.00),v40,z0,tPen\WObj:=wPaper;
    MoveL Offs(pOrigin,396.35,98.22,0.00),v40,z0,tPen\WObj:=wPaper;
    MoveL Offs(pOrigin,396.93,98.54,0.00),v40,z0,tPen\WObj:=wPaper;
    MoveL Offs(pOrigin,397.83,99.44,0.00),v40,z0,tPen\WObj:=wPaper;
    MoveL Offs(pOrigin,396.94,100.04,0.00),v40,z0,tPen\WObj:=wPaper;
    MoveL Offs(pOrigin,396.03,99.14,0.00),v40,z0,tPen\WObj:=wPaper;
    MoveL Offs(pOrigin,394.99,99.58,0.00),v40,z0,tPen\WObj:=wPaper;
    MoveL Offs(pOrigin,395.89,100.49,0.00),v40,z0,tPen\WObj:=wPaper;
    MoveL Offs(pOrigin,396.49,101.06,0.00),v40,z0,tPen\WObj:=wPaper;
    MoveL Offs(pOrigin,403.56,94.00,0.00),v40,z0,tPen\WObj:=wPaper;
    MoveL Offs(pOrigin,404.49,93.61,0.00),v40,z0,tPen\WObj:=wPaper;
    MoveL Offs(pOrigin,400.66,97.01,0.00),v40,z0,tPen\WObj:=wPaper;
    MoveL Offs(pOrigin,399.81,97.44,0.00),v40,z0,tPen\WObj:=wPaper;
    MoveL Offs(pOrigin,400.10,97.30,0.00),v40,z0,tPen\WObj:=wPaper;
    MoveL Offs(pOrigin,396.84,99.42,0.00),v40,z0,tPen\WObj:=wPaper;
    MoveL Offs(pOrigin,393.86,100.77,0.00),v40,z0,tPen\WObj:=wPaper;
    MoveL Offs(pOrigin,392.80,101.76,0.00),v40,z0,tPen\WObj:=wPaper;
    MoveL Offs(pOrigin,388.12,103.39,0.00),v40,z0,tPen\WObj:=wPaper;
    MoveL Offs(pOrigin,380.05,105.09,0.00),v40,z0,tPen\WObj:=wPaper;
    MoveL Offs(pOrigin,373.25,105.30,0.00),v40,z0,tPen\WObj:=wPaper;
    MoveL Offs(pOrigin,369.21,104.66,0.00),v40,z0,tPen\WObj:=wPaper;
    MoveL Offs(pOrigin,365.60,103.39,0.00),v40,z0,tPen\WObj:=wPaper;
    MoveL Offs(pOrigin,361.77,100.41,0.00),v40,z0,tPen\WObj:=wPaper;
    MoveL Offs(pOrigin,359.37,96.80,0.00),v40,z0,tPen\WObj:=wPaper;
    MoveL Offs(pOrigin,359.01,95.53,0.00),v40,fine,tPen\WObj:=wPaper;
    MoveL Offs(pOrigin,359.01,95.53,6.00),v60,z5,tPen\WObj:=wPaper;
    MoveL Offs(pOrigin,360.25,96.98,6.00),vTravel,z5,tPen\WObj:=wPaper;
    MoveL Offs(pOrigin,360.25,96.98,0.00),v60,z0,tPen\WObj:=wPaper;
    MoveL Offs(pOrigin,359.20,98.03,0.00),v40,z0,tPen\WObj:=wPaper;
    MoveL Offs(pOrigin,359.80,98.93,0.00),v40,z0,tPen\WObj:=wPaper;
    MoveL Offs(pOrigin,361.00,97.72,0.00),v40,z0,tPen\WObj:=wPaper;
    MoveL Offs(pOrigin,361.75,98.47,0.00),v40,z0,tPen\WObj:=wPaper;
    MoveL Offs(pOrigin,360.25,99.97,0.00),v40,z0,tPen\WObj:=wPaper;
    MoveL Offs(pOrigin,360.98,99.93,0.00),v40,z0,tPen\WObj:=wPaper;
    MoveL Offs(pOrigin,363.84,102.78,0.00),v40,z0,tPen\WObj:=wPaper;
    MoveL Offs(pOrigin,363.23,102.96,0.00),v40,z0,tPen\WObj:=wPaper;
    MoveL Offs(pOrigin,365.03,101.16,0.00),v40,z0,tPen\WObj:=wPaper;
    MoveL Offs(pOrigin,365.93,101.75,0.00),v40,z0,tPen\WObj:=wPaper;
    MoveL Offs(pOrigin,364.13,103.56,0.00),v40,z0,tPen\WObj:=wPaper;
    MoveL Offs(pOrigin,365.03,104.15,0.00),v40,z0,tPen\WObj:=wPaper;
    MoveL Offs(pOrigin,366.98,102.20,0.00),v40,z0,tPen\WObj:=wPaper;
    MoveL Offs(pOrigin,366.68,102.64,0.00),v40,z0,tPen\WObj:=wPaper;
    MoveL Offs(pOrigin,369.09,105.05,0.00),v40,z0,tPen\WObj:=wPaper;
    MoveL Offs(pOrigin,368.47,105.19,0.00),v40,z0,tPen\WObj:=wPaper;
    MoveL Offs(pOrigin,370.57,103.09,0.00),v40,z0,tPen\WObj:=wPaper;
    MoveL Offs(pOrigin,370.88,103.85,0.00),v40,z0,tPen\WObj:=wPaper;
    MoveL Offs(pOrigin,372.68,105.66,0.00),v40,z0,tPen\WObj:=wPaper;
    MoveL Offs(pOrigin,372.21,105.93,0.00),v40,z0,tPen\WObj:=wPaper;
    MoveL Offs(pOrigin,374.92,103.22,0.00),v40,z0,tPen\WObj:=wPaper;
    MoveL Offs(pOrigin,375.53,104.02,0.00),v40,z0,tPen\WObj:=wPaper;
    MoveL Offs(pOrigin,377.18,105.67,0.00),v40,z0,tPen\WObj:=wPaper;
    MoveL Offs(pOrigin,376.55,106.07,0.00),v40,z0,tPen\WObj:=wPaper;
    MoveL Offs(pOrigin,379.56,103.06,0.00),v40,z0,tPen\WObj:=wPaper;
    MoveL Offs(pOrigin,379.87,103.88,0.00),v40,z0,tPen\WObj:=wPaper;
    MoveL Offs(pOrigin,381.22,105.23,0.00),v40,z0,tPen\WObj:=wPaper;
    MoveL Offs(pOrigin,381.50,105.60,0.00),v40,z0,tPen\WObj:=wPaper;
    MoveL Offs(pOrigin,384.96,102.15,0.00),v40,z0,tPen\WObj:=wPaper;
    MoveL Offs(pOrigin,384.96,103.00,0.00),v40,z0,tPen\WObj:=wPaper;
    MoveL Offs(pOrigin,386.16,104.20,0.00),v40,z0,tPen\WObj:=wPaper;
    MoveL Offs(pOrigin,387.20,104.39,0.00),v40,z0,tPen\WObj:=wPaper;
    MoveL Offs(pOrigin,391.55,100.03,0.00),v40,z0,tPen\WObj:=wPaper;
    MoveL Offs(pOrigin,391.69,100.77,0.00),v40,z0,tPen\WObj:=wPaper;
    MoveL Offs(pOrigin,392.90,101.97,0.00),v40,z0,tPen\WObj:=wPaper;
    MoveL Offs(pOrigin,393.64,102.42,0.00),v40,z0,tPen\WObj:=wPaper;
    MoveL Offs(pOrigin,399.95,96.11,0.00),v40,fine,tPen\WObj:=wPaper;
    MoveL Offs(pOrigin,399.95,96.11,6.00),v60,z5,tPen\WObj:=wPaper;
  ENDPROC

  PROC DrawPart79()
    MoveL Offs(pOrigin,400.70,98.35,6.00),vTravel,z5,tPen\WObj:=wPaper;
    MoveL Offs(pOrigin,400.70,98.35,0.00),v60,z0,tPen\WObj:=wPaper;
    MoveL Offs(pOrigin,404.15,94.90,0.00),v40,fine,tPen\WObj:=wPaper;
    MoveL Offs(pOrigin,404.15,94.90,6.00),v60,z5,tPen\WObj:=wPaper;
    MoveL Offs(pOrigin,405.50,95.04,6.00),vTravel,z5,tPen\WObj:=wPaper;
    MoveL Offs(pOrigin,405.50,95.04,0.00),v60,z0,tPen\WObj:=wPaper;
    MoveL Offs(pOrigin,410.46,90.08,0.00),v40,fine,tPen\WObj:=wPaper;
    MoveL Offs(pOrigin,410.46,90.08,6.00),v60,z5,tPen\WObj:=wPaper;
    MoveL Offs(pOrigin,409.16,91.03,6.00),vTravel,z5,tPen\WObj:=wPaper;
    MoveL Offs(pOrigin,409.16,91.03,0.00),v60,z0,tPen\WObj:=wPaper;
    MoveL Offs(pOrigin,407.67,91.03,0.00),v40,z0,tPen\WObj:=wPaper;
    MoveL Offs(pOrigin,407.46,92.09,0.00),v40,z0,tPen\WObj:=wPaper;
    MoveL Offs(pOrigin,408.95,92.09,0.00),v40,fine,tPen\WObj:=wPaper;
    MoveL Offs(pOrigin,408.95,92.09,6.00),v60,z5,tPen\WObj:=wPaper;
    MoveL Offs(pOrigin,408.69,90.42,6.00),vTravel,z5,tPen\WObj:=wPaper;
    MoveL Offs(pOrigin,408.69,90.42,0.00),v60,z0,tPen\WObj:=wPaper;
    MoveL Offs(pOrigin,408.69,89.15,0.00),v40,fine,tPen\WObj:=wPaper;
    MoveL Offs(pOrigin,408.69,89.15,6.00),v60,z5,tPen\WObj:=wPaper;
    MoveL Offs(pOrigin,407.17,88.89,6.00),vTravel,z5,tPen\WObj:=wPaper;
    MoveL Offs(pOrigin,407.17,88.89,0.00),v60,z0,tPen\WObj:=wPaper;
    MoveL Offs(pOrigin,411.97,84.09,0.00),v40,fine,tPen\WObj:=wPaper;
    MoveL Offs(pOrigin,411.97,84.09,6.00),v60,z5,tPen\WObj:=wPaper;
    MoveL Offs(pOrigin,412.90,80.17,6.00),vTravel,z5,tPen\WObj:=wPaper;
    MoveL Offs(pOrigin,412.90,80.17,0.00),v60,z0,tPen\WObj:=wPaper;
    MoveL Offs(pOrigin,410.95,78.21,0.00),v40,fine,tPen\WObj:=wPaper;
    MoveL Offs(pOrigin,410.95,78.21,6.00),v60,z5,tPen\WObj:=wPaper;
    MoveL Offs(pOrigin,410.86,79.42,6.00),vTravel,z5,tPen\WObj:=wPaper;
    MoveL Offs(pOrigin,410.86,79.42,0.00),v60,z0,tPen\WObj:=wPaper;
    MoveL Offs(pOrigin,412.56,79.42,0.00),v40,z0,tPen\WObj:=wPaper;
    MoveL Offs(pOrigin,413.34,79.74,0.00),v40,z0,tPen\WObj:=wPaper;
    MoveL Offs(pOrigin,407.93,85.15,0.00),v40,fine,tPen\WObj:=wPaper;
    MoveL Offs(pOrigin,407.93,85.15,6.00),v60,z5,tPen\WObj:=wPaper;
    MoveL Offs(pOrigin,410.91,88.13,6.00),vTravel,z5,tPen\WObj:=wPaper;
    MoveL Offs(pOrigin,410.91,88.13,0.00),v60,z0,tPen\WObj:=wPaper;
    MoveL Offs(pOrigin,406.11,92.94,0.00),v40,z0,tPen\WObj:=wPaper;
    MoveL Offs(pOrigin,406.50,93.18,0.00),v40,z0,tPen\WObj:=wPaper;
    MoveL Offs(pOrigin,408.45,95.13,0.00),v40,z0,tPen\WObj:=wPaper;
    MoveL Offs(pOrigin,408.52,94.20,0.00),v40,z0,tPen\WObj:=wPaper;
    MoveL Offs(pOrigin,406.83,94.20,0.00),v40,z0,tPen\WObj:=wPaper;
    MoveL Offs(pOrigin,406.36,94.53,0.00),v40,z0,tPen\WObj:=wPaper;
    MoveL Offs(pOrigin,408.31,96.48,0.00),v40,z0,tPen\WObj:=wPaper;
    MoveL Offs(pOrigin,408.79,96.23,0.00),v40,z0,tPen\WObj:=wPaper;
    MoveL Offs(pOrigin,393.16,111.86,0.00),v40,z0,tPen\WObj:=wPaper;
    MoveL Offs(pOrigin,393.22,111.26,0.00),v40,z0,tPen\WObj:=wPaper;
    MoveL Offs(pOrigin,392.02,110.06,0.00),v40,z0,tPen\WObj:=wPaper;
    MoveL Offs(pOrigin,393.07,109.61,0.00),v40,z0,tPen\WObj:=wPaper;
    MoveL Offs(pOrigin,394.27,110.82,0.00),v40,fine,tPen\WObj:=wPaper;
    MoveL Offs(pOrigin,394.27,110.82,6.00),v60,z5,tPen\WObj:=wPaper;
    MoveL Offs(pOrigin,396.37,109.92,6.00),vTravel,z5,tPen\WObj:=wPaper;
    MoveL Offs(pOrigin,396.37,109.92,0.00),v60,z0,tPen\WObj:=wPaper;
    MoveL Offs(pOrigin,395.01,108.57,0.00),v40,z0,tPen\WObj:=wPaper;
    MoveL Offs(pOrigin,395.91,107.98,0.00),v40,z0,tPen\WObj:=wPaper;
    MoveL Offs(pOrigin,397.26,109.33,0.00),v40,z0,tPen\WObj:=wPaper;
    MoveL Offs(pOrigin,398.26,109.74,0.00),v40,z0,tPen\WObj:=wPaper;
    MoveL Offs(pOrigin,406.23,101.78,0.00),v40,z0,tPen\WObj:=wPaper;
    MoveL Offs(pOrigin,405.33,102.46,0.00),v40,z0,tPen\WObj:=wPaper;
    MoveL Offs(pOrigin,403.53,100.66,0.00),v40,z0,tPen\WObj:=wPaper;
    MoveL Offs(pOrigin,403.85,100.84,0.00),v40,z0,tPen\WObj:=wPaper;
    MoveL Offs(pOrigin,403.64,101.26,0.00),v40,z0,tPen\WObj:=wPaper;
    MoveL Offs(pOrigin,403.85,100.84,0.00),v40,z0,tPen\WObj:=wPaper;
    MoveL Offs(pOrigin,404.28,100.54,0.00),v40,z0,tPen\WObj:=wPaper;
    MoveL Offs(pOrigin,405.76,100.54,0.00),v40,z0,tPen\WObj:=wPaper;
    MoveL Offs(pOrigin,406.37,100.52,0.00),v40,z0,tPen\WObj:=wPaper;
    MoveL Offs(pOrigin,404.57,98.71,0.00),v40,z0,tPen\WObj:=wPaper;
    MoveL Offs(pOrigin,404.91,98.93,0.00),v40,z0,tPen\WObj:=wPaper;
    MoveL Offs(pOrigin,404.70,99.35,0.00),v40,z0,tPen\WObj:=wPaper;
    MoveL Offs(pOrigin,404.91,98.93,0.00),v40,z0,tPen\WObj:=wPaper;
    MoveL Offs(pOrigin,405.34,98.42,0.00),v40,z0,tPen\WObj:=wPaper;
    MoveL Offs(pOrigin,406.83,98.42,0.00),v40,fine,tPen\WObj:=wPaper;
    MoveL Offs(pOrigin,406.83,98.42,6.00),v60,z5,tPen\WObj:=wPaper;
    MoveL Offs(pOrigin,406.19,96.31,6.00),vTravel,z5,tPen\WObj:=wPaper;
    MoveL Offs(pOrigin,406.19,96.31,0.00),v60,z0,tPen\WObj:=wPaper;
    MoveL Offs(pOrigin,407.67,96.31,0.00),v40,fine,tPen\WObj:=wPaper;
    MoveL Offs(pOrigin,407.67,96.31,6.00),v60,z5,tPen\WObj:=wPaper;
    MoveL Offs(pOrigin,408.90,94.08,6.00),vTravel,z5,tPen\WObj:=wPaper;
    MoveL Offs(pOrigin,408.90,94.08,0.00),v60,z0,tPen\WObj:=wPaper;
    MoveL Offs(pOrigin,406.95,92.13,0.00),v40,fine,tPen\WObj:=wPaper;
    MoveL Offs(pOrigin,406.95,92.13,6.00),v60,z5,tPen\WObj:=wPaper;
    MoveL Offs(pOrigin,409.40,94.13,6.00),vTravel,z5,tPen\WObj:=wPaper;
    MoveL Offs(pOrigin,409.40,94.13,0.00),v60,z0,tPen\WObj:=wPaper;
    MoveL Offs(pOrigin,402.79,100.74,0.00),v40,fine,tPen\WObj:=wPaper;
    MoveL Offs(pOrigin,402.79,100.74,6.00),v60,z5,tPen\WObj:=wPaper;
    MoveL Offs(pOrigin,402.79,102.54,6.00),vTravel,z5,tPen\WObj:=wPaper;
    MoveL Offs(pOrigin,402.79,102.54,0.00),v60,z0,tPen\WObj:=wPaper;
    MoveL Offs(pOrigin,403.00,102.11,0.00),v40,z0,tPen\WObj:=wPaper;
    MoveL Offs(pOrigin,402.79,102.54,0.00),v40,fine,tPen\WObj:=wPaper;
    MoveL Offs(pOrigin,402.79,102.54,6.00),v60,z5,tPen\WObj:=wPaper;
    MoveL Offs(pOrigin,401.94,103.60,6.00),vTravel,z5,tPen\WObj:=wPaper;
    MoveL Offs(pOrigin,401.94,103.60,0.00),v60,z0,tPen\WObj:=wPaper;
    MoveL Offs(pOrigin,402.15,103.18,0.00),v40,z0,tPen\WObj:=wPaper;
    MoveL Offs(pOrigin,401.94,103.60,0.00),v40,z0,tPen\WObj:=wPaper;
    MoveL Offs(pOrigin,401.30,104.24,0.00),v40,z0,tPen\WObj:=wPaper;
    MoveL Offs(pOrigin,401.51,103.81,0.00),v40,z0,tPen\WObj:=wPaper;
    MoveL Offs(pOrigin,401.30,104.24,0.00),v40,z0,tPen\WObj:=wPaper;
    MoveL Offs(pOrigin,400.84,103.95,0.00),v40,z0,tPen\WObj:=wPaper;
    MoveL Offs(pOrigin,402.80,105.90,0.00),v40,z0,tPen\WObj:=wPaper;
    MoveL Offs(pOrigin,402.15,105.82,0.00),v40,z0,tPen\WObj:=wPaper;
    MoveL Offs(pOrigin,399.39,105.82,0.00),v40,z0,tPen\WObj:=wPaper;
    MoveL Offs(pOrigin,399.35,105.44,0.00),v40,z0,tPen\WObj:=wPaper;
    MoveL Offs(pOrigin,402.05,108.14,0.00),v40,z0,tPen\WObj:=wPaper;
    MoveL Offs(pOrigin,401.51,107.93,0.00),v40,z0,tPen\WObj:=wPaper;
    MoveL Offs(pOrigin,399.60,107.93,0.00),v40,z0,tPen\WObj:=wPaper;
    MoveL Offs(pOrigin,400.24,108.28,0.00),v40,z0,tPen\WObj:=wPaper;
    MoveL Offs(pOrigin,400.24,105.72,0.00),v40,fine,tPen\WObj:=wPaper;
    MoveL Offs(pOrigin,400.24,105.72,6.00),v60,z5,tPen\WObj:=wPaper;
    MoveL Offs(pOrigin,401.29,104.88,6.00),vTravel,z5,tPen\WObj:=wPaper;
    MoveL Offs(pOrigin,401.29,104.88,0.00),v60,z0,tPen\WObj:=wPaper;
    MoveL Offs(pOrigin,401.29,107.42,0.00),v40,fine,tPen\WObj:=wPaper;
    MoveL Offs(pOrigin,401.29,107.42,6.00),v60,z5,tPen\WObj:=wPaper;
    MoveL Offs(pOrigin,401.30,108.98,6.00),vTravel,z5,tPen\WObj:=wPaper;
    MoveL Offs(pOrigin,401.30,108.98,0.00),v60,z0,tPen\WObj:=wPaper;
    MoveL Offs(pOrigin,399.81,108.98,0.00),v40,z0,tPen\WObj:=wPaper;
    MoveL Offs(pOrigin,399.06,109.63,0.00),v40,z0,tPen\WObj:=wPaper;
    MoveL Offs(pOrigin,401.02,111.59,0.00),v40,z0,tPen\WObj:=wPaper;
    MoveL Offs(pOrigin,400.66,111.10,0.00),v40,z0,tPen\WObj:=wPaper;
    MoveL Offs(pOrigin,399.17,111.10,0.00),v40,z0,tPen\WObj:=wPaper;
    MoveL Offs(pOrigin,398.77,110.83,0.00),v40,z0,tPen\WObj:=wPaper;
    MoveL Offs(pOrigin,400.57,112.63,0.00),v40,z0,tPen\WObj:=wPaper;
    MoveL Offs(pOrigin,400.24,112.15,0.00),v40,z0,tPen\WObj:=wPaper;
    MoveL Offs(pOrigin,398.75,112.15,0.00),v40,z0,tPen\WObj:=wPaper;
  ENDPROC

  PROC DrawPart80()
    MoveL Offs(pOrigin,398.32,111.88,0.00),v40,z0,tPen\WObj:=wPaper;
    MoveL Offs(pOrigin,399.97,113.53,0.00),v40,z0,tPen\WObj:=wPaper;
    MoveL Offs(pOrigin,399.81,113.38,0.00),v40,z0,tPen\WObj:=wPaper;
    MoveL Offs(pOrigin,399.60,113.80,0.00),v40,z0,tPen\WObj:=wPaper;
    MoveL Offs(pOrigin,399.81,113.38,0.00),v40,z0,tPen\WObj:=wPaper;
    MoveL Offs(pOrigin,399.60,113.21,0.00),v40,z0,tPen\WObj:=wPaper;
    MoveL Offs(pOrigin,398.11,113.21,0.00),v40,z0,tPen\WObj:=wPaper;
    MoveL Offs(pOrigin,397.72,112.77,0.00),v40,z0,tPen\WObj:=wPaper;
    MoveL Offs(pOrigin,399.53,114.58,0.00),v40,z0,tPen\WObj:=wPaper;
    MoveL Offs(pOrigin,398.96,114.26,0.00),v40,z0,tPen\WObj:=wPaper;
    MoveL Offs(pOrigin,397.48,114.26,0.00),v40,z0,tPen\WObj:=wPaper;
    MoveL Offs(pOrigin,397.28,113.82,0.00),v40,z0,tPen\WObj:=wPaper;
    MoveL Offs(pOrigin,398.93,115.48,0.00),v40,z0,tPen\WObj:=wPaper;
    MoveL Offs(pOrigin,398.33,115.32,0.00),v40,z0,tPen\WObj:=wPaper;
    MoveL Offs(pOrigin,396.84,115.32,0.00),v40,z0,tPen\WObj:=wPaper;
    MoveL Offs(pOrigin,396.84,115.07,0.00),v40,z0,tPen\WObj:=wPaper;
    MoveL Offs(pOrigin,396.62,115.50,0.00),v40,z0,tPen\WObj:=wPaper;
    MoveL Offs(pOrigin,396.84,115.07,0.00),v40,z0,tPen\WObj:=wPaper;
    MoveL Offs(pOrigin,396.68,114.72,0.00),v40,z0,tPen\WObj:=wPaper;
    MoveL Offs(pOrigin,398.18,116.22,0.00),v40,z0,tPen\WObj:=wPaper;
    MoveL Offs(pOrigin,398.11,116.14,0.00),v40,z0,tPen\WObj:=wPaper;
    MoveL Offs(pOrigin,398.33,115.71,0.00),v40,z0,tPen\WObj:=wPaper;
    MoveL Offs(pOrigin,398.11,116.14,0.00),v40,z0,tPen\WObj:=wPaper;
    MoveL Offs(pOrigin,397.48,116.38,0.00),v40,z0,tPen\WObj:=wPaper;
    MoveL Offs(pOrigin,396.20,116.38,0.00),v40,z0,tPen\WObj:=wPaper;
    MoveL Offs(pOrigin,395.49,116.51,0.00),v40,z0,tPen\WObj:=wPaper;
    MoveL Offs(pOrigin,397.14,118.17,0.00),v40,z0,tPen\WObj:=wPaper;
    MoveL Offs(pOrigin,396.62,118.49,0.00),v40,z0,tPen\WObj:=wPaper;
    MoveL Offs(pOrigin,395.35,118.49,0.00),v40,z0,tPen\WObj:=wPaper;
    MoveL Offs(pOrigin,394.75,118.76,0.00),v40,z0,tPen\WObj:=wPaper;
    MoveL Offs(pOrigin,397.00,121.01,0.00),v40,z0,tPen\WObj:=wPaper;
    MoveL Offs(pOrigin,397.48,120.98,0.00),v40,z0,tPen\WObj:=wPaper;
    MoveL Offs(pOrigin,394.33,124.14,0.00),v40,z0,tPen\WObj:=wPaper;
    MoveL Offs(pOrigin,394.76,124.75,0.00),v40,z0,tPen\WObj:=wPaper;
    MoveL Offs(pOrigin,396.72,126.70,0.00),v40,z0,tPen\WObj:=wPaper;
    MoveL Offs(pOrigin,396.41,126.55,0.00),v40,z0,tPen\WObj:=wPaper;
    MoveL Offs(pOrigin,396.20,126.97,0.00),v40,z0,tPen\WObj:=wPaper;
    MoveL Offs(pOrigin,396.41,126.55,0.00),v40,z0,tPen\WObj:=wPaper;
    MoveL Offs(pOrigin,395.99,126.94,0.00),v40,z0,tPen\WObj:=wPaper;
    MoveL Offs(pOrigin,388.98,126.94,0.00),v40,fine,tPen\WObj:=wPaper;
    MoveL Offs(pOrigin,388.98,126.94,6.00),v60,z5,tPen\WObj:=wPaper;
    MoveL Offs(pOrigin,389.83,127.99,6.00),vTravel,z5,tPen\WObj:=wPaper;
    MoveL Offs(pOrigin,389.83,127.99,0.00),v60,z0,tPen\WObj:=wPaper;
    MoveL Offs(pOrigin,394.92,127.99,0.00),v40,z0,tPen\WObj:=wPaper;
    MoveL Offs(pOrigin,395.35,128.04,0.00),v40,z0,tPen\WObj:=wPaper;
    MoveL Offs(pOrigin,396.48,126.76,0.00),v40,z0,tPen\WObj:=wPaper;
    MoveL Offs(pOrigin,396.84,125.49,0.00),v40,z0,tPen\WObj:=wPaper;
    MoveL Offs(pOrigin,396.62,119.11,0.00),v40,z0,tPen\WObj:=wPaper;
    MoveL Offs(pOrigin,397.83,116.35,0.00),v40,z0,tPen\WObj:=wPaper;
    MoveL Offs(pOrigin,399.88,113.59,0.00),v40,z0,tPen\WObj:=wPaper;
    MoveL Offs(pOrigin,402.72,104.88,0.00),v40,z0,tPen\WObj:=wPaper;
    MoveL Offs(pOrigin,403.99,103.60,0.00),v40,z0,tPen\WObj:=wPaper;
    MoveL Offs(pOrigin,406.12,100.41,0.00),v40,z0,tPen\WObj:=wPaper;
    MoveL Offs(pOrigin,407.75,96.80,0.00),v40,z0,tPen\WObj:=wPaper;
    MoveL Offs(pOrigin,410.86,84.69,0.00),v40,z0,tPen\WObj:=wPaper;
    MoveL Offs(pOrigin,415.33,72.79,0.00),v40,z0,tPen\WObj:=wPaper;
    MoveL Offs(pOrigin,415.96,69.81,0.00),v40,z0,tPen\WObj:=wPaper;
    MoveL Offs(pOrigin,415.75,63.22,0.00),v40,z0,tPen\WObj:=wPaper;
    MoveL Offs(pOrigin,416.60,58.12,0.00),v40,z0,tPen\WObj:=wPaper;
    MoveL Offs(pOrigin,416.39,54.09,0.00),v40,z0,tPen\WObj:=wPaper;
    MoveL Offs(pOrigin,415.75,50.90,0.00),v40,z0,tPen\WObj:=wPaper;
    MoveL Offs(pOrigin,414.33,46.86,0.00),v40,z0,tPen\WObj:=wPaper;
    MoveL Offs(pOrigin,412.35,43.67,0.00),v40,z0,tPen\WObj:=wPaper;
    MoveL Offs(pOrigin,410.86,41.97,0.00),v40,z0,tPen\WObj:=wPaper;
    MoveL Offs(pOrigin,407.89,39.78,0.00),v40,z0,tPen\WObj:=wPaper;
    MoveL Offs(pOrigin,404.49,38.08,0.00),v40,z0,tPen\WObj:=wPaper;
    MoveL Offs(pOrigin,399.60,36.45,0.00),v40,z0,tPen\WObj:=wPaper;
    MoveL Offs(pOrigin,385.58,33.47,0.00),v40,z0,tPen\WObj:=wPaper;
    MoveL Offs(pOrigin,364.11,30.71,0.00),v40,z0,tPen\WObj:=wPaper;
    MoveL Offs(pOrigin,358.38,28.87,0.00),v40,z0,tPen\WObj:=wPaper;
    MoveL Offs(pOrigin,350.51,25.33,0.00),v40,z0,tPen\WObj:=wPaper;
    MoveL Offs(pOrigin,345.20,23.91,0.00),v40,z0,tPen\WObj:=wPaper;
    MoveL Offs(pOrigin,340.10,24.12,0.00),v40,z0,tPen\WObj:=wPaper;
    MoveL Offs(pOrigin,337.34,24.90,0.00),v40,z0,tPen\WObj:=wPaper;
    MoveL Offs(pOrigin,333.30,26.67,0.00),v40,z0,tPen\WObj:=wPaper;
    MoveL Offs(pOrigin,331.81,26.67,0.00),v40,z0,tPen\WObj:=wPaper;
    MoveL Offs(pOrigin,320.34,24.76,0.00),v40,z0,tPen\WObj:=wPaper;
    MoveL Offs(pOrigin,317.79,24.98,0.00),v40,z0,tPen\WObj:=wPaper;
    MoveL Offs(pOrigin,312.69,26.89,0.00),v40,z0,tPen\WObj:=wPaper;
    MoveL Offs(pOrigin,306.74,24.98,0.00),v40,z0,tPen\WObj:=wPaper;
    MoveL Offs(pOrigin,302.06,24.34,0.00),v40,z0,tPen\WObj:=wPaper;
    MoveL Offs(pOrigin,298.24,24.34,0.00),v40,z0,tPen\WObj:=wPaper;
    MoveL Offs(pOrigin,293.14,24.98,0.00),v40,z0,tPen\WObj:=wPaper;
    MoveL Offs(pOrigin,285.91,23.06,0.00),v40,z0,tPen\WObj:=wPaper;
    MoveL Offs(pOrigin,282.30,22.64,0.00),v40,z0,tPen\WObj:=wPaper;
    MoveL Offs(pOrigin,278.05,22.85,0.00),v40,z0,tPen\WObj:=wPaper;
    MoveL Offs(pOrigin,236.19,11.80,0.00),v40,z0,tPen\WObj:=wPaper;
    MoveL Offs(pOrigin,230.45,11.59,0.00),v40,z0,tPen\WObj:=wPaper;
    MoveL Offs(pOrigin,213.24,13.50,0.00),v40,z0,tPen\WObj:=wPaper;
    MoveL Offs(pOrigin,207.50,13.07,0.00),v40,z0,tPen\WObj:=wPaper;
    MoveL Offs(pOrigin,196.45,14.14,0.00),v40,z0,tPen\WObj:=wPaper;
    MoveL Offs(pOrigin,194.96,14.49,0.00),v40,z0,tPen\WObj:=wPaper;
    MoveL Offs(pOrigin,193.69,15.41,0.00),v40,z0,tPen\WObj:=wPaper;
    MoveL Offs(pOrigin,106.35,24.55,0.00),v40,z0,tPen\WObj:=wPaper;
    MoveL Offs(pOrigin,87.44,26.25,0.00),v40,z0,tPen\WObj:=wPaper;
    MoveL Offs(pOrigin,86.16,26.53,0.00),v40,z0,tPen\WObj:=wPaper;
    MoveL Offs(pOrigin,85.17,27.52,0.00),v40,z0,tPen\WObj:=wPaper;
    MoveL Offs(pOrigin,84.89,28.38,0.00),v40,z0,tPen\WObj:=wPaper;
    MoveL Offs(pOrigin,85.10,31.77,0.00),v40,z0,tPen\WObj:=wPaper;
    MoveL Offs(pOrigin,86.80,33.33,0.00),v40,z0,tPen\WObj:=wPaper;
    MoveL Offs(pOrigin,92.32,34.96,0.00),v40,z0,tPen\WObj:=wPaper;
    MoveL Offs(pOrigin,107.62,38.58,0.00),v40,z0,tPen\WObj:=wPaper;
    MoveL Offs(pOrigin,107.73,37.72,0.00),v40,z0,tPen\WObj:=wPaper;
    MoveL Offs(pOrigin,107.73,41.34,0.00),v40,z0,tPen\WObj:=wPaper;
    MoveL Offs(pOrigin,108.26,41.40,0.00),v40,z0,tPen\WObj:=wPaper;
    MoveL Offs(pOrigin,106.56,41.40,0.00),v40,z0,tPen\WObj:=wPaper;
    MoveL Offs(pOrigin,106.56,41.12,0.00),v40,z0,tPen\WObj:=wPaper;
    MoveL Offs(pOrigin,106.14,41.76,0.00),v40,z0,tPen\WObj:=wPaper;
    MoveL Offs(pOrigin,106.56,41.12,0.00),v40,z0,tPen\WObj:=wPaper;
    MoveL Offs(pOrigin,106.14,40.34,0.00),v40,z0,tPen\WObj:=wPaper;
    MoveL Offs(pOrigin,109.75,40.34,0.00),v40,z0,tPen\WObj:=wPaper;
    MoveL Offs(pOrigin,109.96,40.49,0.00),v40,z0,tPen\WObj:=wPaper;
    MoveL Offs(pOrigin,110.39,40.28,0.00),v40,z0,tPen\WObj:=wPaper;
    MoveL Offs(pOrigin,109.96,40.49,0.00),v40,z0,tPen\WObj:=wPaper;
    MoveL Offs(pOrigin,109.54,40.70,0.00),v40,z0,tPen\WObj:=wPaper;
    MoveL Offs(pOrigin,110.60,39.99,0.00),v40,z0,tPen\WObj:=wPaper;
    MoveL Offs(pOrigin,111.66,39.85,0.00),v40,z0,tPen\WObj:=wPaper;
    MoveL Offs(pOrigin,111.95,39.85,0.00),v40,z0,tPen\WObj:=wPaper;
    MoveL Offs(pOrigin,111.95,38.15,0.00),v40,z0,tPen\WObj:=wPaper;
    MoveL Offs(pOrigin,113.01,38.15,0.00),v40,z0,tPen\WObj:=wPaper;
  ENDPROC

  PROC DrawPart81()
    MoveL Offs(pOrigin,113.01,39.85,0.00),v40,z0,tPen\WObj:=wPaper;
    MoveL Offs(pOrigin,113.58,40.34,0.00),v40,z0,tPen\WObj:=wPaper;
    MoveL Offs(pOrigin,111.66,40.34,0.00),v40,z0,tPen\WObj:=wPaper;
    MoveL Offs(pOrigin,110.89,39.64,0.00),v40,z0,tPen\WObj:=wPaper;
    MoveL Offs(pOrigin,110.89,37.94,0.00),v40,z0,tPen\WObj:=wPaper;
    MoveL Offs(pOrigin,111.52,37.15,0.00),v40,z0,tPen\WObj:=wPaper;
    MoveL Offs(pOrigin,117.38,43.01,0.00),v40,z0,tPen\WObj:=wPaper;
    MoveL Offs(pOrigin,116.97,42.40,0.00),v40,z0,tPen\WObj:=wPaper;
    MoveL Offs(pOrigin,116.76,43.25,0.00),v40,z0,tPen\WObj:=wPaper;
    MoveL Offs(pOrigin,115.91,43.67,0.00),v40,z0,tPen\WObj:=wPaper;
    MoveL Offs(pOrigin,115.91,43.67,0.00),v40,z0,tPen\WObj:=wPaper;
    MoveL Offs(pOrigin,115.49,44.95,0.00),v40,z0,tPen\WObj:=wPaper;
    MoveL Offs(pOrigin,114.00,44.74,0.00),v40,z0,tPen\WObj:=wPaper;
    MoveL Offs(pOrigin,113.36,45.16,0.00),v40,z0,tPen\WObj:=wPaper;
    MoveL Offs(pOrigin,111.88,44.95,0.00),v40,z0,tPen\WObj:=wPaper;
    MoveL Offs(pOrigin,111.88,44.95,0.00),v40,z0,tPen\WObj:=wPaper;
    MoveL Offs(pOrigin,112.30,43.89,0.00),v40,z0,tPen\WObj:=wPaper;
    MoveL Offs(pOrigin,112.30,43.89,0.00),v40,z0,tPen\WObj:=wPaper;
    MoveL Offs(pOrigin,112.30,42.19,0.00),v40,z0,tPen\WObj:=wPaper;
    MoveL Offs(pOrigin,111.66,41.76,0.00),v40,z0,tPen\WObj:=wPaper;
    MoveL Offs(pOrigin,111.66,41.76,0.00),v40,z0,tPen\WObj:=wPaper;
    MoveL Offs(pOrigin,111.10,42.19,0.00),v40,z0,tPen\WObj:=wPaper;
    MoveL Offs(pOrigin,110.60,43.89,0.00),v40,z0,tPen\WObj:=wPaper;
    MoveL Offs(pOrigin,111.03,44.88,0.00),v40,z0,tPen\WObj:=wPaper;
    MoveL Offs(pOrigin,111.88,44.95,0.00),v40,z0,tPen\WObj:=wPaper;
    MoveL Offs(pOrigin,112.15,45.24,0.00),v40,z0,tPen\WObj:=wPaper;
    MoveL Offs(pOrigin,110.65,43.74,0.00),v40,z0,tPen\WObj:=wPaper;
    MoveL Offs(pOrigin,109.95,44.12,0.00),v40,z0,tPen\WObj:=wPaper;
    MoveL Offs(pOrigin,118.52,35.55,0.00),v40,fine,tPen\WObj:=wPaper;
    MoveL Offs(pOrigin,118.52,35.55,6.00),v60,z5,tPen\WObj:=wPaper;
    MoveL Offs(pOrigin,117.61,36.45,6.00),vTravel,z5,tPen\WObj:=wPaper;
    MoveL Offs(pOrigin,117.61,36.45,0.00),v60,z0,tPen\WObj:=wPaper;
    MoveL Offs(pOrigin,116.97,36.66,0.00),v40,z0,tPen\WObj:=wPaper;
    MoveL Offs(pOrigin,115.06,36.03,0.00),v40,z0,tPen\WObj:=wPaper;
    MoveL Offs(pOrigin,96.57,33.47,0.00),v40,fine,tPen\WObj:=wPaper;
    MoveL Offs(pOrigin,96.57,33.47,6.00),v60,z5,tPen\WObj:=wPaper;
    MoveL Offs(pOrigin,97.13,31.71,6.00),vTravel,z5,tPen\WObj:=wPaper;
    MoveL Offs(pOrigin,97.13,31.71,0.00),v60,z0,tPen\WObj:=wPaper;
    MoveL Offs(pOrigin,91.27,25.85,0.00),v40,z0,tPen\WObj:=wPaper;
    MoveL Offs(pOrigin,91.43,25.30,0.00),v40,z0,tPen\WObj:=wPaper;
    MoveL Offs(pOrigin,84.67,32.06,0.00),v40,z0,tPen\WObj:=wPaper;
    MoveL Offs(pOrigin,84.99,31.52,0.00),v40,z0,tPen\WObj:=wPaper;
    MoveL Offs(pOrigin,87.25,33.78,0.00),v40,z0,tPen\WObj:=wPaper;
    MoveL Offs(pOrigin,87.06,34.15,0.00),v40,z0,tPen\WObj:=wPaper;
    MoveL Offs(pOrigin,96.38,24.84,0.00),v40,z0,tPen\WObj:=wPaper;
    MoveL Offs(pOrigin,95.61,25.71,0.00),v40,z0,tPen\WObj:=wPaper;
    MoveL Offs(pOrigin,101.17,31.27,0.00),v40,z0,tPen\WObj:=wPaper;
    MoveL Offs(pOrigin,101.45,31.71,0.00),v40,z0,tPen\WObj:=wPaper;
    MoveL Offs(pOrigin,109.87,23.30,0.00),v40,fine,tPen\WObj:=wPaper;
    MoveL Offs(pOrigin,109.87,23.30,6.00),v60,z5,tPen\WObj:=wPaper;
    MoveL Offs(pOrigin,111.88,27.67,6.00),vTravel,z5,tPen\WObj:=wPaper;
    MoveL Offs(pOrigin,111.88,27.67,0.00),v60,z0,tPen\WObj:=wPaper;
    MoveL Offs(pOrigin,107.84,27.67,0.00),v40,fine,tPen\WObj:=wPaper;
    MoveL Offs(pOrigin,107.84,27.67,6.00),v60,z5,tPen\WObj:=wPaper;
    MoveL Offs(pOrigin,107.41,29.23,6.00),vTravel,z5,tPen\WObj:=wPaper;
    MoveL Offs(pOrigin,107.41,29.23,0.00),v60,z0,tPen\WObj:=wPaper;
    MoveL Offs(pOrigin,106.78,29.65,0.00),v40,z0,tPen\WObj:=wPaper;
    MoveL Offs(pOrigin,105.07,29.44,0.00),v40,z0,tPen\WObj:=wPaper;
    MoveL Offs(pOrigin,104.44,29.86,0.00),v40,z0,tPen\WObj:=wPaper;
    MoveL Offs(pOrigin,102.53,29.65,0.00),v40,z0,tPen\WObj:=wPaper;
    MoveL Offs(pOrigin,102.53,29.65,0.00),v40,z0,tPen\WObj:=wPaper;
    MoveL Offs(pOrigin,101.89,28.87,0.00),v40,z0,tPen\WObj:=wPaper;
    MoveL Offs(pOrigin,88.29,30.08,0.00),v40,z0,tPen\WObj:=wPaper;
    MoveL Offs(pOrigin,86.66,30.71,0.00),v40,z0,tPen\WObj:=wPaper;
    MoveL Offs(pOrigin,86.80,31.49,0.00),v40,z0,tPen\WObj:=wPaper;
    MoveL Offs(pOrigin,89.14,31.77,0.00),v40,z0,tPen\WObj:=wPaper;
    MoveL Offs(pOrigin,89.78,32.41,0.00),v40,z0,tPen\WObj:=wPaper;
    MoveL Offs(pOrigin,90.41,33.05,0.00),v40,z0,tPen\WObj:=wPaper;
    MoveL Offs(pOrigin,100.40,35.60,0.00),v40,z0,tPen\WObj:=wPaper;
    MoveL Offs(pOrigin,111.03,37.51,0.00),v40,z0,tPen\WObj:=wPaper;
    MoveL Offs(pOrigin,125.26,39.00,0.00),v40,z0,tPen\WObj:=wPaper;
    MoveL Offs(pOrigin,128.02,39.00,0.00),v40,z0,tPen\WObj:=wPaper;
    MoveL Offs(pOrigin,128.88,38.72,0.00),v40,z0,tPen\WObj:=wPaper;
    MoveL Offs(pOrigin,129.09,38.15,0.00),v40,z0,tPen\WObj:=wPaper;
    MoveL Offs(pOrigin,129.09,38.15,0.00),v40,z0,tPen\WObj:=wPaper;
    MoveL Offs(pOrigin,127.81,37.94,0.00),v40,z0,tPen\WObj:=wPaper;
    MoveL Offs(pOrigin,127.39,37.30,0.00),v40,z0,tPen\WObj:=wPaper;
    MoveL Offs(pOrigin,127.39,37.30,0.00),v40,z0,tPen\WObj:=wPaper;
    MoveL Offs(pOrigin,126.96,36.88,0.00),v40,z0,tPen\WObj:=wPaper;
    MoveL Offs(pOrigin,125.26,37.09,0.00),v40,z0,tPen\WObj:=wPaper;
    MoveL Offs(pOrigin,125.26,37.09,0.00),v40,z0,tPen\WObj:=wPaper;
    MoveL Offs(pOrigin,124.84,36.66,0.00),v40,z0,tPen\WObj:=wPaper;
    MoveL Offs(pOrigin,123.35,36.88,0.00),v40,z0,tPen\WObj:=wPaper;
    MoveL Offs(pOrigin,123.35,36.88,0.00),v40,z0,tPen\WObj:=wPaper;
    MoveL Offs(pOrigin,122.71,36.45,0.00),v40,z0,tPen\WObj:=wPaper;
    MoveL Offs(pOrigin,121.86,36.52,0.00),v40,z0,tPen\WObj:=wPaper;
    MoveL Offs(pOrigin,121.65,36.88,0.00),v40,z0,tPen\WObj:=wPaper;
    MoveL Offs(pOrigin,122.29,37.30,0.00),v40,z0,tPen\WObj:=wPaper;
    MoveL Offs(pOrigin,123.35,37.30,0.00),v40,z0,tPen\WObj:=wPaper;
    MoveL Offs(pOrigin,123.35,37.30,0.00),v40,z0,tPen\WObj:=wPaper;
    MoveL Offs(pOrigin,125.26,37.51,0.00),v40,z0,tPen\WObj:=wPaper;
    MoveL Offs(pOrigin,125.26,37.51,0.00),v40,z0,tPen\WObj:=wPaper;
    MoveL Offs(pOrigin,127.39,37.72,0.00),v40,z0,tPen\WObj:=wPaper;
    MoveL Offs(pOrigin,127.39,37.30,0.00),v40,z0,tPen\WObj:=wPaper;
    MoveL Offs(pOrigin,133.55,37.09,0.00),v40,z0,tPen\WObj:=wPaper;
    MoveL Offs(pOrigin,146.30,35.60,0.00),v40,z0,tPen\WObj:=wPaper;
    MoveL Offs(pOrigin,149.06,35.60,0.00),v40,z0,tPen\WObj:=wPaper;
    MoveL Offs(pOrigin,153.52,36.45,0.00),v40,z0,tPen\WObj:=wPaper;
    MoveL Offs(pOrigin,154.59,36.24,0.00),v40,z0,tPen\WObj:=wPaper;
    MoveL Offs(pOrigin,155.01,36.45,0.00),v40,z0,tPen\WObj:=wPaper;
    MoveL Offs(pOrigin,155.23,37.09,0.00),v40,z0,tPen\WObj:=wPaper;
    MoveL Offs(pOrigin,155.25,36.88,0.00),v40,z0,tPen\WObj:=wPaper;
    MoveL Offs(pOrigin,155.25,38.15,0.00),v40,z0,tPen\WObj:=wPaper;
    MoveL Offs(pOrigin,155.86,38.23,0.00),v40,z0,tPen\WObj:=wPaper;
    MoveL Offs(pOrigin,147.36,38.23,0.00),v40,z0,tPen\WObj:=wPaper;
    MoveL Offs(pOrigin,147.85,39.00,0.00),v40,z0,tPen\WObj:=wPaper;
    MoveL Offs(pOrigin,147.85,41.12,0.00),v40,z0,tPen\WObj:=wPaper;
    MoveL Offs(pOrigin,148.21,41.40,0.00),v40,z0,tPen\WObj:=wPaper;
    MoveL Offs(pOrigin,141.62,41.40,0.00),v40,z0,tPen\WObj:=wPaper;
    MoveL Offs(pOrigin,141.20,41.55,0.00),v40,z0,tPen\WObj:=wPaper;
    MoveL Offs(pOrigin,140.35,42.40,0.00),v40,z0,tPen\WObj:=wPaper;
    MoveL Offs(pOrigin,141.20,41.55,0.00),v40,z0,tPen\WObj:=wPaper;
    MoveL Offs(pOrigin,141.05,41.28,0.00),v40,z0,tPen\WObj:=wPaper;
    MoveL Offs(pOrigin,144.65,44.89,0.00),v40,z0,tPen\WObj:=wPaper;
    MoveL Offs(pOrigin,144.18,44.57,0.00),v40,z0,tPen\WObj:=wPaper;
    MoveL Offs(pOrigin,138.86,44.57,0.00),v40,z0,tPen\WObj:=wPaper;
    MoveL Offs(pOrigin,139.41,44.52,0.00),v40,z0,tPen\WObj:=wPaper;
    MoveL Offs(pOrigin,139.41,47.08,0.00),v40,z0,tPen\WObj:=wPaper;
    MoveL Offs(pOrigin,139.00,47.57,0.00),v40,z0,tPen\WObj:=wPaper;
    MoveL Offs(pOrigin,139.29,48.14,0.00),v40,z0,tPen\WObj:=wPaper;
  ENDPROC

  PROC DrawPart82()
    MoveL Offs(pOrigin,139.29,50.05,0.00),v40,z0,tPen\WObj:=wPaper;
    MoveL Offs(pOrigin,138.65,50.47,0.00),v40,z0,tPen\WObj:=wPaper;
    MoveL Offs(pOrigin,138.08,50.05,0.00),v40,z0,tPen\WObj:=wPaper;
    MoveL Offs(pOrigin,138.01,49.41,0.00),v40,z0,tPen\WObj:=wPaper;
    MoveL Offs(pOrigin,138.37,48.14,0.00),v40,z0,tPen\WObj:=wPaper;
    MoveL Offs(pOrigin,139.00,47.57,0.00),v40,fine,tPen\WObj:=wPaper;
    MoveL Offs(pOrigin,139.00,47.57,6.00),v60,z5,tPen\WObj:=wPaper;
    MoveL Offs(pOrigin,139.50,48.79,6.00),vTravel,z5,tPen\WObj:=wPaper;
    MoveL Offs(pOrigin,139.50,48.79,0.00),v60,z0,tPen\WObj:=wPaper;
    MoveL Offs(pOrigin,143.11,48.79,0.00),v40,z0,tPen\WObj:=wPaper;
    MoveL Offs(pOrigin,143.62,48.33,0.00),v40,z0,tPen\WObj:=wPaper;
    MoveL Offs(pOrigin,138.96,43.67,0.00),v40,z0,tPen\WObj:=wPaper;
    MoveL Offs(pOrigin,139.71,43.51,0.00),v40,z0,tPen\WObj:=wPaper;
    MoveL Offs(pOrigin,145.02,43.51,0.00),v40,z0,tPen\WObj:=wPaper;
    MoveL Offs(pOrigin,144.69,43.25,0.00),v40,z0,tPen\WObj:=wPaper;
    MoveL Offs(pOrigin,144.69,39.85,0.00),v40,z0,tPen\WObj:=wPaper;
    MoveL Offs(pOrigin,144.39,39.29,0.00),v40,z0,tPen\WObj:=wPaper;
    MoveL Offs(pOrigin,153.95,39.29,0.00),v40,z0,tPen\WObj:=wPaper;
    MoveL Offs(pOrigin,154.19,38.79,0.00),v40,z0,tPen\WObj:=wPaper;
    MoveL Offs(pOrigin,154.19,36.88,0.00),v40,z0,tPen\WObj:=wPaper;
    MoveL Offs(pOrigin,153.91,36.23,0.00),v40,z0,tPen\WObj:=wPaper;
    MoveL Offs(pOrigin,156.32,38.63,0.00),v40,z0,tPen\WObj:=wPaper;
    MoveL Offs(pOrigin,155.86,38.58,0.00),v40,z0,tPen\WObj:=wPaper;
    MoveL Offs(pOrigin,155.65,38.79,0.00),v40,z0,tPen\WObj:=wPaper;
    MoveL Offs(pOrigin,155.86,38.36,0.00),v40,z0,tPen\WObj:=wPaper;
    MoveL Offs(pOrigin,157.14,38.36,0.00),v40,z0,tPen\WObj:=wPaper;
    MoveL Offs(pOrigin,157.22,38.04,0.00),v40,z0,tPen\WObj:=wPaper;
    MoveL Offs(pOrigin,155.26,36.08,0.00),v40,z0,tPen\WObj:=wPaper;
    MoveL Offs(pOrigin,155.23,36.45,0.00),v40,z0,tPen\WObj:=wPaper;
    MoveL Offs(pOrigin,157.77,35.67,0.00),v40,z0,tPen\WObj:=wPaper;
    MoveL Offs(pOrigin,159.90,34.11,0.00),v40,z0,tPen\WObj:=wPaper;
    MoveL Offs(pOrigin,159.60,34.45,0.00),v40,z0,tPen\WObj:=wPaper;
    MoveL Offs(pOrigin,160.65,35.50,0.00),v40,z0,tPen\WObj:=wPaper;
    MoveL Offs(pOrigin,160.75,35.06,0.00),v40,z0,tPen\WObj:=wPaper;
    MoveL Offs(pOrigin,158.84,35.06,0.00),v40,z0,tPen\WObj:=wPaper;
    MoveL Offs(pOrigin,158.70,35.04,0.00),v40,z0,tPen\WObj:=wPaper;
    MoveL Offs(pOrigin,159.76,36.10,0.00),v40,z0,tPen\WObj:=wPaper;
    MoveL Offs(pOrigin,158.84,36.12,0.00),v40,z0,tPen\WObj:=wPaper;
    MoveL Offs(pOrigin,155.86,36.12,0.00),v40,z0,tPen\WObj:=wPaper;
    MoveL Offs(pOrigin,156.46,35.79,0.00),v40,z0,tPen\WObj:=wPaper;
    MoveL Offs(pOrigin,158.11,37.44,0.00),v40,z0,tPen\WObj:=wPaper;
    MoveL Offs(pOrigin,157.56,37.18,0.00),v40,z0,tPen\WObj:=wPaper;
    MoveL Offs(pOrigin,149.70,37.18,0.00),v40,fine,tPen\WObj:=wPaper;
    MoveL Offs(pOrigin,149.70,37.18,6.00),v60,z5,tPen\WObj:=wPaper;
    MoveL Offs(pOrigin,150.47,35.77,6.00),vTravel,z5,tPen\WObj:=wPaper;
    MoveL Offs(pOrigin,150.47,35.77,0.00),v60,z0,tPen\WObj:=wPaper;
    MoveL Offs(pOrigin,154.37,39.68,0.00),v40,z0,tPen\WObj:=wPaper;
    MoveL Offs(pOrigin,155.27,39.08,0.00),v40,z0,tPen\WObj:=wPaper;
    MoveL Offs(pOrigin,152.27,36.07,0.00),v40,z0,tPen\WObj:=wPaper;
    MoveL Offs(pOrigin,151.61,36.12,0.00),v40,z0,tPen\WObj:=wPaper;
    MoveL Offs(pOrigin,141.84,36.12,0.00),v40,z0,tPen\WObj:=wPaper;
    MoveL Offs(pOrigin,141.78,36.04,0.00),v40,z0,tPen\WObj:=wPaper;
    MoveL Offs(pOrigin,147.79,42.05,0.00),v40,z0,tPen\WObj:=wPaper;
    MoveL Offs(pOrigin,146.80,41.55,0.00),v40,z0,tPen\WObj:=wPaper;
    MoveL Offs(pOrigin,146.80,39.21,0.00),v40,z0,tPen\WObj:=wPaper;
    MoveL Offs(pOrigin,145.74,39.42,0.00),v40,z0,tPen\WObj:=wPaper;
    MoveL Offs(pOrigin,145.74,42.19,0.00),v40,z0,tPen\WObj:=wPaper;
    MoveL Offs(pOrigin,146.09,42.46,0.00),v40,z0,tPen\WObj:=wPaper;
    MoveL Offs(pOrigin,140.56,42.46,0.00),v40,z0,tPen\WObj:=wPaper;
    MoveL Offs(pOrigin,140.30,42.03,0.00),v40,z0,tPen\WObj:=wPaper;
    MoveL Offs(pOrigin,144.21,45.94,0.00),v40,z0,tPen\WObj:=wPaper;
    MoveL Offs(pOrigin,143.75,45.62,0.00),v40,z0,tPen\WObj:=wPaper;
    MoveL Offs(pOrigin,138.01,45.62,0.00),v40,z0,tPen\WObj:=wPaper;
    MoveL Offs(pOrigin,137.61,45.32,0.00),v40,z0,tPen\WObj:=wPaper;
    MoveL Offs(pOrigin,143.93,51.63,0.00),v40,z0,tPen\WObj:=wPaper;
    MoveL Offs(pOrigin,144.23,51.65,0.00),v40,z0,tPen\WObj:=wPaper;
    MoveL Offs(pOrigin,136.57,59.32,0.00),v40,z0,tPen\WObj:=wPaper;
    MoveL Offs(pOrigin,137.17,60.21,0.00),v40,z0,tPen\WObj:=wPaper;
    MoveL Offs(pOrigin,144.68,52.70,0.00),v40,z0,tPen\WObj:=wPaper;
    MoveL Offs(pOrigin,144.23,53.43,0.00),v40,z0,tPen\WObj:=wPaper;
    MoveL Offs(pOrigin,137.17,46.36,0.00),v40,z0,tPen\WObj:=wPaper;
    MoveL Offs(pOrigin,137.16,46.44,0.00),v40,z0,tPen\WObj:=wPaper;
    MoveL Offs(pOrigin,137.16,47.29,0.00),v40,z0,tPen\WObj:=wPaper;
    MoveL Offs(pOrigin,135.89,50.90,0.00),v40,z0,tPen\WObj:=wPaper;
    MoveL Offs(pOrigin,136.10,55.79,0.00),v40,z0,tPen\WObj:=wPaper;
    MoveL Offs(pOrigin,136.88,58.12,0.00),v40,z0,tPen\WObj:=wPaper;
    MoveL Offs(pOrigin,138.01,60.04,0.00),v40,z0,tPen\WObj:=wPaper;
    MoveL Offs(pOrigin,142.26,64.71,0.00),v40,z0,tPen\WObj:=wPaper;
    MoveL Offs(pOrigin,148.00,68.82,0.00),v40,z0,tPen\WObj:=wPaper;
    MoveL Offs(pOrigin,150.34,70.10,0.00),v40,z0,tPen\WObj:=wPaper;
    MoveL Offs(pOrigin,154.16,71.51,0.00),v40,z0,tPen\WObj:=wPaper;
    MoveL Offs(pOrigin,156.29,71.94,0.00),v40,z0,tPen\WObj:=wPaper;
    MoveL Offs(pOrigin,159.90,71.94,0.00),v40,z0,tPen\WObj:=wPaper;
    MoveL Offs(pOrigin,166.49,69.60,0.00),v40,z0,tPen\WObj:=wPaper;
    MoveL Offs(pOrigin,166.91,69.81,0.00),v40,z0,tPen\WObj:=wPaper;
    MoveL Offs(pOrigin,167.12,70.45,0.00),v40,z0,tPen\WObj:=wPaper;
    MoveL Offs(pOrigin,166.27,71.09,0.00),v40,z0,tPen\WObj:=wPaper;
    MoveL Offs(pOrigin,166.49,70.97,0.00),v40,z0,tPen\WObj:=wPaper;
    MoveL Offs(pOrigin,171.38,70.97,0.00),v40,z0,tPen\WObj:=wPaper;
    MoveL Offs(pOrigin,171.09,71.51,0.00),v40,z0,tPen\WObj:=wPaper;
    MoveL Offs(pOrigin,171.09,72.79,0.00),v40,z0,tPen\WObj:=wPaper;
    MoveL Offs(pOrigin,170.52,73.21,0.00),v40,z0,tPen\WObj:=wPaper;
    MoveL Offs(pOrigin,170.10,73.64,0.00),v40,z0,tPen\WObj:=wPaper;
    MoveL Offs(pOrigin,170.52,73.21,0.00),v40,z0,tPen\WObj:=wPaper;
    MoveL Offs(pOrigin,170.03,73.21,0.00),v40,z0,tPen\WObj:=wPaper;
    MoveL Offs(pOrigin,170.03,70.88,0.00),v40,z0,tPen\WObj:=wPaper;
    MoveL Offs(pOrigin,170.10,69.91,0.00),v40,z0,tPen\WObj:=wPaper;
    MoveL Offs(pOrigin,166.70,69.91,0.00),v40,fine,tPen\WObj:=wPaper;
    MoveL Offs(pOrigin,166.70,69.91,6.00),v60,z5,tPen\WObj:=wPaper;
    MoveL Offs(pOrigin,167.92,70.66,6.00),vTravel,z5,tPen\WObj:=wPaper;
    MoveL Offs(pOrigin,167.92,70.66,0.00),v60,z0,tPen\WObj:=wPaper;
    MoveL Offs(pOrigin,167.92,68.96,0.00),v40,z0,tPen\WObj:=wPaper;
    MoveL Offs(pOrigin,168.82,68.86,0.00),v40,z0,tPen\WObj:=wPaper;
    MoveL Offs(pOrigin,148.85,68.86,0.00),v40,z0,tPen\WObj:=wPaper;
    MoveL Offs(pOrigin,148.91,68.75,0.00),v40,z0,tPen\WObj:=wPaper;
    MoveL Offs(pOrigin,148.91,66.41,0.00),v40,z0,tPen\WObj:=wPaper;
    MoveL Offs(pOrigin,149.97,66.84,0.00),v40,z0,tPen\WObj:=wPaper;
    MoveL Offs(pOrigin,149.97,69.18,0.00),v40,z0,tPen\WObj:=wPaper;
    MoveL Offs(pOrigin,150.76,69.91,0.00),v40,z0,tPen\WObj:=wPaper;
    MoveL Offs(pOrigin,165.00,69.91,0.00),v40,z0,tPen\WObj:=wPaper;
    MoveL Offs(pOrigin,164.75,69.60,0.00),v40,z0,tPen\WObj:=wPaper;
    MoveL Offs(pOrigin,164.75,68.54,0.00),v40,z0,tPen\WObj:=wPaper;
    MoveL Offs(pOrigin,164.35,67.57,0.00),v40,z0,tPen\WObj:=wPaper;
    MoveL Offs(pOrigin,170.66,73.88,0.00),v40,z0,tPen\WObj:=wPaper;
    MoveL Offs(pOrigin,169.68,74.14,0.00),v40,z0,tPen\WObj:=wPaper;
    MoveL Offs(pOrigin,149.28,74.14,0.00),v40,z0,tPen\WObj:=wPaper;
    MoveL Offs(pOrigin,149.39,75.01,0.00),v40,z0,tPen\WObj:=wPaper;
    MoveL Offs(pOrigin,146.54,72.16,0.00),v40,z0,tPen\WObj:=wPaper;
    MoveL Offs(pOrigin,146.72,71.57,0.00),v40,z0,tPen\WObj:=wPaper;
    MoveL Offs(pOrigin,144.31,73.97,0.00),v40,z0,tPen\WObj:=wPaper;
  ENDPROC

  PROC DrawPart83()
    MoveL Offs(pOrigin,145.34,73.95,0.00),v40,z0,tPen\WObj:=wPaper;
    MoveL Offs(pOrigin,141.89,70.50,0.00),v40,z0,tPen\WObj:=wPaper;
    MoveL Offs(pOrigin,142.05,70.97,0.00),v40,z0,tPen\WObj:=wPaper;
    MoveL Offs(pOrigin,139.50,70.97,0.00),v40,z0,tPen\WObj:=wPaper;
    MoveL Offs(pOrigin,139.71,69.91,0.00),v40,z0,tPen\WObj:=wPaper;
    MoveL Offs(pOrigin,136.95,69.91,0.00),v40,z0,tPen\WObj:=wPaper;
    MoveL Offs(pOrigin,137.38,68.86,0.00),v40,z0,tPen\WObj:=wPaper;
    MoveL Offs(pOrigin,134.61,68.86,0.00),v40,fine,tPen\WObj:=wPaper;
    MoveL Offs(pOrigin,134.61,68.86,6.00),v60,z5,tPen\WObj:=wPaper;
    MoveL Offs(pOrigin,133.69,69.66,6.00),vTravel,z5,tPen\WObj:=wPaper;
    MoveL Offs(pOrigin,133.69,69.66,0.00),v60,z0,tPen\WObj:=wPaper;
    MoveL Offs(pOrigin,136.10,67.26,0.00),v40,z0,tPen\WObj:=wPaper;
    MoveL Offs(pOrigin,135.88,67.48,0.00),v40,z0,tPen\WObj:=wPaper;
    MoveL Offs(pOrigin,140.69,72.29,0.00),v40,z0,tPen\WObj:=wPaper;
    MoveL Offs(pOrigin,141.02,72.78,0.00),v40,z0,tPen\WObj:=wPaper;
    MoveL Offs(pOrigin,143.43,70.38,0.00),v40,z0,tPen\WObj:=wPaper;
    MoveL Offs(pOrigin,144.47,70.83,0.00),v40,z0,tPen\WObj:=wPaper;
    MoveL Offs(pOrigin,142.07,73.23,0.00),v40,z0,tPen\WObj:=wPaper;
    MoveL Offs(pOrigin,143.12,73.68,0.00),v40,z0,tPen\WObj:=wPaper;
    MoveL Offs(pOrigin,145.52,71.27,0.00),v40,z0,tPen\WObj:=wPaper;
    MoveL Offs(pOrigin,145.02,72.02,0.00),v40,z0,tPen\WObj:=wPaper;
    MoveL Offs(pOrigin,142.05,72.02,0.00),v40,fine,tPen\WObj:=wPaper;
    MoveL Offs(pOrigin,142.05,72.02,6.00),v60,z5,tPen\WObj:=wPaper;
    MoveL Offs(pOrigin,143.24,73.35,6.00),vTravel,z5,tPen\WObj:=wPaper;
    MoveL Offs(pOrigin,143.24,73.35,0.00),v60,z0,tPen\WObj:=wPaper;
    MoveL Offs(pOrigin,139.34,69.44,0.00),v40,z0,tPen\WObj:=wPaper;
    MoveL Offs(pOrigin,139.09,68.75,0.00),v40,z0,tPen\WObj:=wPaper;
    MoveL Offs(pOrigin,136.68,71.15,0.00),v40,z0,tPen\WObj:=wPaper;
    MoveL Offs(pOrigin,135.64,70.70,0.00),v40,z0,tPen\WObj:=wPaper;
    MoveL Offs(pOrigin,138.19,68.15,0.00),v40,z0,tPen\WObj:=wPaper;
    MoveL Offs(pOrigin,137.14,67.70,0.00),v40,z0,tPen\WObj:=wPaper;
    MoveL Offs(pOrigin,134.74,70.11,0.00),v40,z0,tPen\WObj:=wPaper;
    MoveL Offs(pOrigin,135.59,70.18,0.00),v40,z0,tPen\WObj:=wPaper;
    MoveL Offs(pOrigin,125.83,60.41,0.00),v40,z0,tPen\WObj:=wPaper;
    MoveL Offs(pOrigin,126.96,60.25,0.00),v40,z0,tPen\WObj:=wPaper;
    MoveL Offs(pOrigin,127.39,60.67,0.00),v40,z0,tPen\WObj:=wPaper;
    MoveL Offs(pOrigin,126.96,60.25,0.00),v40,z0,tPen\WObj:=wPaper;
    MoveL Offs(pOrigin,127.39,60.67,0.00),v40,z0,tPen\WObj:=wPaper;
    MoveL Offs(pOrigin,127.53,61.74,0.00),v40,z0,tPen\WObj:=wPaper;
    MoveL Offs(pOrigin,128.45,63.65,0.00),v40,z0,tPen\WObj:=wPaper;
    MoveL Offs(pOrigin,128.45,63.65,0.00),v40,z0,tPen\WObj:=wPaper;
    MoveL Offs(pOrigin,130.15,64.29,0.00),v40,z0,tPen\WObj:=wPaper;
    MoveL Offs(pOrigin,130.15,64.29,0.00),v40,z0,tPen\WObj:=wPaper;
    MoveL Offs(pOrigin,129.87,63.01,0.00),v40,z0,tPen\WObj:=wPaper;
    MoveL Offs(pOrigin,128.59,61.31,0.00),v40,z0,tPen\WObj:=wPaper;
    MoveL Offs(pOrigin,127.39,60.67,0.00),v40,z0,tPen\WObj:=wPaper;
    MoveL Offs(pOrigin,127.39,60.67,0.00),v40,z0,tPen\WObj:=wPaper;
    MoveL Offs(pOrigin,126.11,58.34,0.00),v40,z0,tPen\WObj:=wPaper;
    MoveL Offs(pOrigin,126.11,58.34,0.00),v40,z0,tPen\WObj:=wPaper;
    MoveL Offs(pOrigin,125.05,54.51,0.00),v40,z0,tPen\WObj:=wPaper;
    MoveL Offs(pOrigin,125.26,53.24,0.00),v40,z0,tPen\WObj:=wPaper;
    MoveL Offs(pOrigin,125.05,48.56,0.00),v40,z0,tPen\WObj:=wPaper;
    MoveL Offs(pOrigin,125.76,46.01,0.00),v40,z0,tPen\WObj:=wPaper;
    MoveL Offs(pOrigin,127.03,43.75,0.00),v40,z0,tPen\WObj:=wPaper;
    MoveL Offs(pOrigin,128.02,43.46,0.00),v40,z0,tPen\WObj:=wPaper;
    MoveL Offs(pOrigin,128.17,43.34,0.00),v40,z0,tPen\WObj:=wPaper;
    MoveL Offs(pOrigin,123.06,38.23,0.00),v40,z0,tPen\WObj:=wPaper;
    MoveL Offs(pOrigin,122.51,39.21,0.00),v40,z0,tPen\WObj:=wPaper;
    MoveL Offs(pOrigin,122.51,41.76,0.00),v40,z0,tPen\WObj:=wPaper;
    MoveL Offs(pOrigin,122.71,42.46,0.00),v40,z0,tPen\WObj:=wPaper;
    MoveL Offs(pOrigin,120.16,42.46,0.00),v40,z0,tPen\WObj:=wPaper;
    MoveL Offs(pOrigin,120.40,42.19,0.00),v40,z0,tPen\WObj:=wPaper;
    MoveL Offs(pOrigin,120.40,47.08,0.00),v40,z0,tPen\WObj:=wPaper;
    MoveL Offs(pOrigin,121.01,46.68,0.00),v40,z0,tPen\WObj:=wPaper;
    MoveL Offs(pOrigin,119.52,46.68,0.00),v40,z0,tPen\WObj:=wPaper;
    MoveL Offs(pOrigin,119.19,46.31,0.00),v40,z0,tPen\WObj:=wPaper;
    MoveL Offs(pOrigin,121.45,48.56,0.00),v40,z0,tPen\WObj:=wPaper;
    MoveL Offs(pOrigin,121.77,48.73,0.00),v40,z0,tPen\WObj:=wPaper;
    MoveL Offs(pOrigin,118.77,51.73,0.00),v40,z0,tPen\WObj:=wPaper;
    MoveL Offs(pOrigin,119.21,52.30,0.00),v40,z0,tPen\WObj:=wPaper;
    MoveL Offs(pOrigin,138.14,71.23,0.00),v40,z0,tPen\WObj:=wPaper;
    MoveL Offs(pOrigin,137.88,71.45,0.00),v40,z0,tPen\WObj:=wPaper;
    MoveL Offs(pOrigin,140.13,69.19,0.00),v40,fine,tPen\WObj:=wPaper;
    MoveL Offs(pOrigin,140.13,69.19,6.00),v60,z5,tPen\WObj:=wPaper;
    MoveL Offs(pOrigin,141.33,69.49,6.00),vTravel,z5,tPen\WObj:=wPaper;
    MoveL Offs(pOrigin,141.33,69.49,0.00),v60,z0,tPen\WObj:=wPaper;
    MoveL Offs(pOrigin,138.93,71.89,0.00),v40,z0,tPen\WObj:=wPaper;
    MoveL Offs(pOrigin,139.98,72.34,0.00),v40,z0,tPen\WObj:=wPaper;
    MoveL Offs(pOrigin,142.38,69.93,0.00),v40,fine,tPen\WObj:=wPaper;
    MoveL Offs(pOrigin,142.38,69.93,6.00),v60,z5,tPen\WObj:=wPaper;
    MoveL Offs(pOrigin,144.29,71.40,6.00),vTravel,z5,tPen\WObj:=wPaper;
    MoveL Offs(pOrigin,144.29,71.40,0.00),v60,z0,tPen\WObj:=wPaper;
    MoveL Offs(pOrigin,147.44,74.56,0.00),v40,z0,tPen\WObj:=wPaper;
    MoveL Offs(pOrigin,147.91,74.86,0.00),v40,z0,tPen\WObj:=wPaper;
    MoveL Offs(pOrigin,150.31,72.46,0.00),v40,z0,tPen\WObj:=wPaper;
    MoveL Offs(pOrigin,150.58,73.22,0.00),v40,z0,tPen\WObj:=wPaper;
    MoveL Offs(pOrigin,152.84,75.47,0.00),v40,z0,tPen\WObj:=wPaper;
    MoveL Offs(pOrigin,152.85,75.89,0.00),v40,z0,tPen\WObj:=wPaper;
    MoveL Offs(pOrigin,161.56,67.18,0.00),v40,z0,tPen\WObj:=wPaper;
    MoveL Offs(pOrigin,161.65,67.86,0.00),v40,z0,tPen\WObj:=wPaper;
    MoveL Offs(pOrigin,169.31,75.52,0.00),v40,z0,tPen\WObj:=wPaper;
    MoveL Offs(pOrigin,169.04,75.19,0.00),v40,z0,tPen\WObj:=wPaper;
    MoveL Offs(pOrigin,167.98,75.19,0.00),v40,fine,tPen\WObj:=wPaper;
    MoveL Offs(pOrigin,167.98,75.19,6.00),v60,z5,tPen\WObj:=wPaper;
    MoveL Offs(pOrigin,168.97,74.49,6.00),vTravel,z5,tPen\WObj:=wPaper;
    MoveL Offs(pOrigin,168.97,74.49,0.00),v60,z0,tPen\WObj:=wPaper;
    MoveL Offs(pOrigin,168.97,72.79,0.00),v40,z0,tPen\WObj:=wPaper;
    MoveL Offs(pOrigin,168.61,72.57,0.00),v40,z0,tPen\WObj:=wPaper;
    MoveL Offs(pOrigin,169.04,72.36,0.00),v40,z0,tPen\WObj:=wPaper;
    MoveL Offs(pOrigin,168.61,72.57,0.00),v40,z0,tPen\WObj:=wPaper;
    MoveL Offs(pOrigin,169.04,72.02,0.00),v40,z0,tPen\WObj:=wPaper;
    MoveL Offs(pOrigin,172.44,72.02,0.00),v40,z0,tPen\WObj:=wPaper;
    MoveL Offs(pOrigin,172.65,71.94,0.00),v40,z0,tPen\WObj:=wPaper;
    MoveL Offs(pOrigin,173.71,73.00,0.00),v40,z0,tPen\WObj:=wPaper;
    MoveL Offs(pOrigin,172.65,71.94,0.00),v40,z0,tPen\WObj:=wPaper;
    MoveL Offs(pOrigin,173.38,71.79,0.00),v40,z0,tPen\WObj:=wPaper;
    MoveL Offs(pOrigin,164.82,80.35,0.00),v40,z0,tPen\WObj:=wPaper;
    MoveL Offs(pOrigin,165.44,80.60,0.00),v40,z0,tPen\WObj:=wPaper;
    MoveL Offs(pOrigin,166.64,81.81,0.00),v40,z0,tPen\WObj:=wPaper;
    MoveL Offs(pOrigin,167.06,82.59,0.00),v40,z0,tPen\WObj:=wPaper;
    MoveL Offs(pOrigin,156.54,93.11,0.00),v40,z0,tPen\WObj:=wPaper;
    MoveL Offs(pOrigin,156.48,92.56,0.00),v40,z0,tPen\WObj:=wPaper;
    MoveL Offs(pOrigin,155.43,91.51,0.00),v40,z0,tPen\WObj:=wPaper;
    MoveL Offs(pOrigin,154.54,92.11,0.00),v40,z0,tPen\WObj:=wPaper;
    MoveL Offs(pOrigin,155.44,93.01,0.00),v40,fine,tPen\WObj:=wPaper;
    MoveL Offs(pOrigin,155.44,93.01,6.00),v60,z5,tPen\WObj:=wPaper;
    MoveL Offs(pOrigin,158.84,92.09,6.00),vTravel,z5,tPen\WObj:=wPaper;
    MoveL Offs(pOrigin,158.84,92.09,0.00),v60,z0,tPen\WObj:=wPaper;
    MoveL Offs(pOrigin,163.73,92.09,0.00),v40,z0,tPen\WObj:=wPaper;
    MoveL Offs(pOrigin,162.64,92.12,0.00),v40,z0,tPen\WObj:=wPaper;
  ENDPROC

